(* CODESYS project Rezka.project
   Company: Plinfa
   Title: Rezka
   Author: Surmylo Serhii
   Version: 0.0.0.0

Project tree, tasks and I/O mapping:
  MyController : TM241CEC24T/U, Schneider Electric, order no. TM241CEC24T/U, version 4.0.2.20
    application Application
      task MAST (cyclic, interval 20 ms, priority 15, watchdog 100 ms x 1) calls POU_outputs_11_20, POU_outputs_21_30, POU_outputs_31_40, POU_outputs_41_50, POU_outputs_51_64, POU_outputs_drivers, POU_10_outputs_oilstation, POU_1_Utils, POU_2_TrosTolkateli, POU_3_PodvodTelezhki, POU_4_Zahvat, POU_6_HorizontalCutting, POU_7_VerticalCutting, POU_9_altivars, POU_5_Oprokidyvanie
      function HiddenPOU [ST]
      global variables GVL
      trace Trace (task MAST): POU.M_K1
      Symbols
      program POU_10_outputs_oilstation [LD]
      program POU_4_Zahvat [LD]
      program POU_1_Utils [LD]
      program POU_outputs_11_20 [LD]
      program POU_outputs_31_40 [LD]
      program POU_outputs_21_30 [LD]
      program POU_outputs_41_50 [LD]
      program POU_outputs_51_64 [LD]
      program POU_3_PodvodTelezhki [LD]
      program POU_2_TrosTolkateli [LD]
      program POU_outputs_drivers [LD]
      program POU_9_altivars [LD]
      program POU_7_VerticalCutting [LD]
      program POU_6_HorizontalCutting [LD]
      program POU_5_Oprokidyvanie [LD]
      program POU_interlock [LD]
      program POU_interlock_double [LD]
      module_unites/
        program PressTable_in [LD]
        program GrabTroll_out [LD]
        program GrabTroll_in [LD]
        program CentrTroll_in [LD]
        program TurnTroll_in [LD]
        program CentrTroll_out [LD]
        program TurnTroll_out [LD]
        program TakeTable_in [LD]
        program TakeTable_out [LD]
        program MoveTipper_in [LD]
        program MoveTipper_out [LD]
        program FixingFrame_in [LD]
        program FixingFrame_out [LD]
        program PressTable_out [LD]
        program CuttingFrame_dn [LD]
        program CuttingFrame_up [LD]
        program MovingFrame_fwd [LD]
        program MovingFrame_rev [LD]
    DI : Digital Inputs, Schneider Electric, version 4.0.2.20
        unmapped channels: IW0, IB1
    DQ : Digital Outputs, Schneider Electric, version 4.0.2.20
        unmapped channels: QW0, QB1
    Counters : Counters, Schneider Electric, version 4.0.2.20
    Pulse_Generators : Pulse Generators, Schneider Electric, version 4.0.2.20
    Cartridge_1 : Cartridge, Schneider Electric, version 4.0.2.20
    IO_Bus : IO bus - TM3, Schneider Electric, version 4.0.2.20
      Module_1 : TM3DI32K, Schneider Electric, order no. TM3DI32K, version 1.0.1.1
          input  idwModule_1_ID0 : DWORD  // ID0
          input  KM2 : BOOL  // ID0.I0
          input  KM3 : BOOL  // ID0.I1
          input  KM4 : BOOL  // ID0.I2
          input  KM7 : BOOL  // ID0.I3
          input  KM8 : BOOL  // ID0.I4
          input  KM9 : BOOL  // ID0.I5
          input  KM10 : BOOL  // ID0.I6
          input  KM11 : BOOL  // ID0.I7
          input  KM12 : BOOL  // ID0.I8
          input  KM13 : BOOL  // ID0.I9
          input  KM14 : BOOL  // ID0.I10
          input  PuskAvt : BOOL  // ID0.I11
          input  Stop : BOOL  // ID0.I12
          input  SQ1_s : BOOL  // ID0.I16
          input  SQ2_s : BOOL  // ID0.I17
          input  Kluch1_s : BOOL  // ID0.I18
          input  Vper1_s : BOOL  // ID0.I19
          input  Naz1_s : BOOL  // ID0.I20
          input  SQ3_s : BOOL  // ID0.I21
          input  SQ4_s : BOOL  // ID0.I22
          input  SQ5_s : BOOL  // ID0.I23
          input  SQ6_s : BOOL  // ID0.I24
          input  HED2_1_s : BOOL  // ID0.I25
          input  HED2_2_s : BOOL  // ID0.I26
          input  HED2_5_s : BOOL  // ID0.I29
      Module_2 : TM3DI32K, Schneider Electric, order no. TM3DI32K, version 1.0.1.1
          input  idwModule_2_ID0 : DWORD  // ID0
          input  C3B_s : BOOL  // ID0.I1
          input  C4B_s : BOOL  // ID0.I2
          input  C5B_s : BOOL  // ID0.I3
          input  C6B_s : BOOL  // ID0.I4
          input  C5C_s : BOOL  // ID0.I5
          input  C6C_s : BOOL  // ID0.I6
          input  C13B_s : BOOL  // ID0.I7
          input  C14B_s : BOOL  // ID0.I8
          input  C13C_s : BOOL  // ID0.I9
          input  C14C_s : BOOL  // ID0.I10
          input  C11B_s : BOOL  // ID0.I11
          input  C12B_s : BOOL  // ID0.I12
          input  C34_s : BOOL  // ID0.I13
          input  C3A_s : BOOL  // ID0.I14
          input  C4A_s : BOOL  // ID0.I15
          input  C5A_s : BOOL  // ID0.I16
          input  C6A_s : BOOL  // ID0.I17
          input  C5D_s : BOOL  // ID0.I18
          input  C6D_s : BOOL  // ID0.I19
          input  C13A_s : BOOL  // ID0.I20
          input  C14A_s : BOOL  // ID0.I21
          input  C13D_s : BOOL  // ID0.I22
          input  C14D_s : BOOL  // ID0.I23
          input  C11A_s : BOOL  // ID0.I24
          input  C12A_s : BOOL  // ID0.I25
          input  C17_s : BOOL  // ID0.I26
          input  C17A_s : BOOL  // ID0.I27
          input  C17B_s : BOOL  // ID0.I28
          input  C18A_s : BOOL  // ID0.I29
          input  C18B_s : BOOL  // ID0.I30
          input  C17C_s : BOOL  // ID0.I31
      Module_3 : TM3DI32K, Schneider Electric, order no. TM3DI32K, version 1.0.1.1
          input  idwModule_3_ID0 : DWORD  // ID0
          input  C17D_s : BOOL  // ID0.I0
          input  C18C_s : BOOL  // ID0.I1
          input  C18D_s : BOOL  // ID0.I2
          input  C16_s : BOOL  // ID0.I3
          input  C21_s : BOOL  // ID0.I4
          input  C22_s : BOOL  // ID0.I5
          input  C28_s : BOOL  // ID0.I6
          input  C29_s : BOOL  // ID0.I7
          input  C30_s : BOOL  // ID0.I8
          input  C31_s : BOOL  // ID0.I9
          input  C32_s : BOOL  // ID0.I10
          input  C2_s : BOOL  // ID0.I11
          input  C2A_s : BOOL  // ID0.I12
          input  C23B_s : BOOL  // ID0.I13
          input  C23C_s : BOOL  // ID0.I14
          input  C7_s : BOOL  // ID0.I15
          input  C8_s : BOOL  // ID0.I16
          input  C9_s : BOOL  // ID0.I17
          input  C15_s : BOOL  // ID0.I18
          input  C19_s : BOOL  // ID0.I19
          input  C20_s : BOOL  // ID0.I20
          input  C27_s : BOOL  // ID0.I21
          input  C33_s : BOOL  // ID0.I22
          input  C35_s : BOOL  // ID0.I23
          input  C1_s : BOOL  // ID0.I24
          input  C1A_s : BOOL  // ID0.I25
          input  C23A_s : BOOL  // ID0.I26
          input  C23D_s : BOOL  // ID0.I27
          input  C25_s : BOOL  // ID0.I28
          input  C26_s : BOOL  // ID0.I29
          input  C10_s : BOOL  // ID0.I31
      Module_4 : TM3DI32K, Schneider Electric, order no. TM3DI32K, version 1.0.1.1
          input  idwModule_4_ID0 : DWORD  // ID0
          input  SQ10_s : BOOL  // ID0.I0
          input  SQ11_s : BOOL  // ID0.I1
          input  Kluch2_s : BOOL  // ID0.I2
          input  Vper2_s : BOOL  // ID0.I3
          input  Naz2_s : BOOL  // ID0.I4
          input  SQ12_s : BOOL  // ID0.I5
          input  SQ13_s : BOOL  // ID0.I6
          input  SQ14_s : BOOL  // ID0.I7
          input  Kluch3_s : BOOL  // ID0.I8
          input  Vper3_s : BOOL  // ID0.I9
          input  Naz3_s : BOOL  // ID0.I10
          input  SQ15_s : BOOL  // ID0.I11
          input  SQ16_s : BOOL  // ID0.I12
          input  SQ17_s : BOOL  // ID0.I13
          input  SQ18_s : BOOL  // ID0.I14
          input  SQ19_s : BOOL  // ID0.I15
          input  C21shtrih_s : BOOL  // ID0.I20
          input  C22shtrih_s : BOOL  // ID0.I21
      Module_5 : TM3DQ32TK, Schneider Electric, order no. TM3DQ32TK, version 1.0.1.1
          output KL1 : BOOL  // QD0.Q0
          output KL2 : BOOL  // QD0.Q1
          output KL3 : BOOL  // QD0.Q2
          output KL4 : BOOL  // QD0.Q3
          output KL5 : BOOL  // QD0.Q4
          output KL6 : BOOL  // QD0.Q5
          output KL7 : BOOL  // QD0.Q6
          output KL8 : BOOL  // QD0.Q7
          output KL9 : BOOL  // QD0.Q8
          output KL10 : BOOL  // QD0.Q9
          output KL11 : BOOL  // QD0.Q10
          output KL12 : BOOL  // QD0.Q11
          output KL13 : BOOL  // QD0.Q12
          output KL14 : BOOL  // QD0.Q13
          output KL15 : BOOL  // QD0.Q14
          output KL16 : BOOL  // QD0.Q15
          output KL17 : BOOL  // QD0.Q16
          output KL18 : BOOL  // QD0.Q17
          output KL19 : BOOL  // QD0.Q18
          output KL20 : BOOL  // QD0.Q19
          output KL21 : BOOL  // QD0.Q20
          output KL22 : BOOL  // QD0.Q21
          output KL23 : BOOL  // QD0.Q22
          output KL24 : BOOL  // QD0.Q23
          output KL25 : BOOL  // QD0.Q24
          output KL26 : BOOL  // QD0.Q25
          output KL27 : BOOL  // QD0.Q26
          output KL28 : BOOL  // QD0.Q27
          output KL29 : BOOL  // QD0.Q28
          output KL30 : BOOL  // QD0.Q29
          output KL31 : BOOL  // QD0.Q30
          output KL32 : BOOL  // QD0.Q31
          unmapped channels: QD0
      Module_6 : TM3DQ32TK, Schneider Electric, order no. TM3DQ32TK, version 1.0.1.1
          output KL33 : BOOL  // QD0.Q0
          output KL34 : BOOL  // QD0.Q1
          output KL35 : BOOL  // QD0.Q2
          output KL36 : BOOL  // QD0.Q3
          output KL37 : BOOL  // QD0.Q4
          output KL38 : BOOL  // QD0.Q5
          output KL39 : BOOL  // QD0.Q6
          output KL40 : BOOL  // QD0.Q7
          output KL41 : BOOL  // QD0.Q8
          output KL42 : BOOL  // QD0.Q9
          output KL43 : BOOL  // QD0.Q10
          output KL44 : BOOL  // QD0.Q11
          output KL45 : BOOL  // QD0.Q12
          output KL46 : BOOL  // QD0.Q13
          output KL47 : BOOL  // QD0.Q14
          output KL48 : BOOL  // QD0.Q15
          output KL49 : BOOL  // QD0.Q16
          output KL50 : BOOL  // QD0.Q17
          output KL51 : BOOL  // QD0.Q18
          output KL52 : BOOL  // QD0.Q19
          output KL53 : BOOL  // QD0.Q20
          output KL54 : BOOL  // QD0.Q21
          output KL55 : BOOL  // QD0.Q22
          output KL56 : BOOL  // QD0.Q23
          output KL57 : BOOL  // QD0.Q24
          output KL58 : BOOL  // QD0.Q25
          output KL59 : BOOL  // QD0.Q26
          output KL60 : BOOL  // QD0.Q27
          output KL61 : BOOL  // QD0.Q28
          output KL62 : BOOL  // QD0.Q29
          output KL63 : BOOL  // QD0.Q30
          output KL64 : BOOL  // QD0.Q31
          unmapped channels: QD0
    COM_Bus : COM bus, Schneider Electric, version 4.0.2.20
    Ethernet_1 : Ethernet Network, Schneider Electric, version 4.0.2.20
        settings: IPAddress = [192, 168, 49, 90]; SubnetMask = [255, 255, 255, 0]; GatewayAddress = [192, 168, 49, 1]; DeviceName = 'sch_cutter'; WebServer = TRUE; FTP Server = FALSE; SoMachine Protocol = TRUE; Modbus Server = TRUE; NetManage Protocol = TRUE; SNMP protocol = TRUE; Enable Routing = FALSE; WebVisu protocol = FALSE
      ModbusTCP_Slave_Device : ModbusTCP Slave Device, Schneider Electric, version 3.5.2.3
          settings: IPMasterAddress = [192, 168, 0, 90]
          unmapped channels: Inputs, Outputs
    Serial_Line_1 : Serial line, Schneider Electric, version 4.0.2.20
      SoMachine_Network_Manager : SoMachine-Network Manager, Schneider Electric, version 4.0.0.2
    Serial_Line_2 : Serial line, Schneider Electric, version 4.0.2.20
      Modbus_Manager : Modbus Manager, Schneider Electric, version 4.0.0.2
    CAN_1 : CANopen bus, Schneider Electric, version 4.0.2.20
      CANopen_Performance : CANopen Performance, Schneider Electric, order no. 1806, version 3.0.1.22
          settings: ConfigVersion = 50659584
        Altivar_71_0 : Altivar 71, Schneider Electric, order no. 71, version 4.4.5.0
            settings: General Options.Optional Device = TRUE; General Options.Reset Node = TRUE; NODEIDSAVED = 1; SDO Timeout = 1000000; Explicit Deactivate PDOs = TRUE; EXPERTSETTINGS = True; Heartbeat-Producer Time = 300; PDO 16#1400.COBID = 16#0201; Settings.COBID = 16#0181; Settings.Transmission Type = 16#FF; Settings.available PDO-Parameter.Inhibit Time available = TRUE; Settings.available PDO-Parameter.Event Timer available = TRUE; Settings.Inhibit Time = 30; Settings.Event Timer = 1000; Generic COBID = '$NODEID+16#0180'; Heartbeat-Consuming1.Heartbeat-Time = 300 ms; Controlword.Subindex = 16#00; Frequency ref..Index = 16#2002; Frequency ref..Subindex = 16#04; Frequency ref..ObjectLength = 16; Motor current.Index = 16#2002; Motor current.Subindex = 16#05; Motor current.ObjectLength = 16; Output frequency.Index = 16#2002; Output frequency.Subindex = 16#03; Output frequency.ObjectLength = 16; Error Code.Index = 16#603F; Error Code.Subindex = 16#00; Error Code.ObjectLength = 16; Statusword.Index = 16#6041; Statusword.Subindex = 16#00; Statusword.ObjectLength = 16; SDO List.Set Guardtime.Index = 16#100C; SDO List.Set Guardtime.Subindex = 16#00; SDO List.Set Guardtime.Value = 16#00000000; SDO List.Set Guardtime.Size = 16; SDO List.Set Guardtime.AbortIfError = FALSE; SDO List.Set Guardtime.JumpToLine = FALSE; SDO List.Set Guardtime.Line = 0; SDO List.Set Lifetime.Index = 16#100D;
              SDO List.Set Lifetime.Subindex = 16#00; SDO List.Set Lifetime.Value = 16#00000000; SDO List.Set Lifetime.Size = 8; SDO List.Set Lifetime.AbortIfError = FALSE; SDO List.Set Lifetime.JumpToLine = FALSE; SDO List.Set Lifetime.Line = 0; SDO List.Set Heartbeat Consumer.Index = 16#1016; SDO List.Set Heartbeat Consumer.Subindex = 16#01; SDO List.Set Heartbeat Consumer.Value = 16#007F012C; SDO List.Set Heartbeat Consumer.Size = 32; SDO List.Set Heartbeat Consumer.AbortIfError = FALSE; SDO List.Set Heartbeat Consumer.JumpToLine = FALSE; SDO List.Set Heartbeat Consumer.Line = 0; SDO List.Set Heartbeat Producer.Index = 16#1017; SDO List.Set Heartbeat Producer.Subindex = 16#00; SDO List.Set Heartbeat Producer.Value = 16#0000012C; SDO List.Set Heartbeat Producer.Size = 16; SDO List.Set Heartbeat Producer.AbortIfError = FALSE; SDO List.Set Heartbeat Producer.JumpToLine = FALSE; SDO List.Set Heartbeat Producer.Line = 0; SDO List.Disable PDO.Index = 16#1400; SDO List.Disable PDO.Subindex = 16#01; SDO List.Disable PDO.Value = 16#80000201; SDO List.Disable PDO.Size = 32; SDO List.Disable PDO.AbortIfError = FALSE; SDO List.Disable PDO.JumpToLine = FALSE; SDO List.Disable PDO.Line = 0; SDO List.Set transmission type.Index = 16#1400; SDO List.Set transmission type.Subindex = 16#02; SDO List.Set transmission type.Value = 16#FF; SDO List.Set transmission type.Size = 8; SDO List.Set transmission type.AbortIfError = FALSE; SDO List.Set transmission type.JumpToLine = FALSE; SDO List.Set transmission type.Line = 0; SDO List.Clear pdo mapping.Index = 16#1600; SDO List.Clear pdo mapping.Subindex = 16#00; SDO List.Clear pdo mapping.Value = 16#0; SDO List.Clear pdo mapping.Size = 8; SDO List.Clear pdo mapping.AbortIfError = FALSE; SDO List.Clear pdo mapping.JumpToLine = FALSE;
              SDO List.Clear pdo mapping.Line = 0; SDO List.Set Mapping.Index = 16#1600; SDO List.Set Mapping.Subindex = 16#01; SDO List.Set Mapping.Value = 16#60400010; SDO List.Set Mapping.Size = 32; SDO List.Set Mapping.AbortIfError = FALSE; SDO List.Set Mapping.JumpToLine = FALSE; SDO List.Set Mapping.Line = 0; SDO List.Set Mapping.Index = 16#1600; SDO List.Set Mapping.Subindex = 16#02; SDO List.Set Mapping.Value = 16#20020410; SDO List.Set Mapping.Size = 32; SDO List.Set Mapping.AbortIfError = FALSE; SDO List.Set Mapping.JumpToLine = FALSE; SDO List.Set Mapping.Line = 0; SDO List.Set Mapping.Index = 16#1600; SDO List.Set Mapping.Subindex = 16#03; SDO List.Set Mapping.Value = 16#20020510; SDO List.Set Mapping.Size = 32; SDO List.Set Mapping.AbortIfError = FALSE; SDO List.Set Mapping.JumpToLine = FALSE; SDO List.Set Mapping.Line = 0; SDO List.Set Mapping.Index = 16#1600; SDO List.Set Mapping.Subindex = 16#04; SDO List.Set Mapping.Value = 16#20020310; SDO List.Set Mapping.Size = 32; SDO List.Set Mapping.AbortIfError = FALSE; SDO List.Set Mapping.JumpToLine = FALSE; SDO List.Set Mapping.Line = 0; SDO List.Set number of pdos.Index = 16#1600; SDO List.Set number of pdos.Subindex = 16#00; SDO List.Set number of pdos.Value = 16#04; SDO List.Set number of pdos.Size = 8; SDO List.Set number of pdos.AbortIfError = FALSE; SDO List.Set number of pdos.JumpToLine = FALSE; SDO List.Set number of pdos.Line = 0; SDO List.Set and enable COB-ID.Index = 16#1400; SDO List.Set and enable COB-ID.Subindex = 16#01; SDO List.Set and enable COB-ID.Value = 16#00000201; SDO List.Set and enable COB-ID.Size = 32;
              SDO List.Set and enable COB-ID.AbortIfError = FALSE; SDO List.Set and enable COB-ID.JumpToLine = FALSE; SDO List.Set and enable COB-ID.Line = 0; SDO List.Disable PDO.Index = 16#1800; SDO List.Disable PDO.Subindex = 16#01; SDO List.Disable PDO.Value = 16#80000181; SDO List.Disable PDO.Size = 32; SDO List.Disable PDO.AbortIfError = FALSE; SDO List.Disable PDO.JumpToLine = FALSE; SDO List.Disable PDO.Line = 0; SDO List.Set transmission type.Index = 16#1800; SDO List.Set transmission type.Subindex = 16#02; SDO List.Set transmission type.Value = 16#FF; SDO List.Set transmission type.Size = 8; SDO List.Set transmission type.AbortIfError = FALSE; SDO List.Set transmission type.JumpToLine = FALSE; SDO List.Set transmission type.Line = 0; SDO List.Set inhibit time.Index = 16#1800; SDO List.Set inhibit time.Subindex = 16#03; SDO List.Set inhibit time.Value = 16#001E; SDO List.Set inhibit time.Size = 16; SDO List.Set inhibit time.AbortIfError = FALSE; SDO List.Set inhibit time.JumpToLine = FALSE; SDO List.Set inhibit time.Line = 0; SDO List.Set event time.Index = 16#1800; SDO List.Set event time.Subindex = 16#05; SDO List.Set event time.Value = 16#03E8; SDO List.Set event time.Size = 16; SDO List.Set event time.AbortIfError = FALSE; SDO List.Set event time.JumpToLine = FALSE; SDO List.Set event time.Line = 0; SDO List.Clear pdo mapping.Index = 16#1A00; SDO List.Clear pdo mapping.Subindex = 16#00; SDO List.Clear pdo mapping.Value = 16#0; SDO List.Clear pdo mapping.Size = 8; SDO List.Clear pdo mapping.AbortIfError = FALSE; SDO List.Clear pdo mapping.JumpToLine = FALSE; SDO List.Clear pdo mapping.Line = 0; SDO List.Set Mapping.Index = 16#1A00; SDO List.Set Mapping.Subindex = 16#01;
              SDO List.Set Mapping.Value = 16#603F0010; SDO List.Set Mapping.Size = 32; SDO List.Set Mapping.AbortIfError = FALSE; SDO List.Set Mapping.JumpToLine = FALSE; SDO List.Set Mapping.Line = 0; SDO List.Set Mapping.Index = 16#1A00; SDO List.Set Mapping.Subindex = 16#02; SDO List.Set Mapping.Value = 16#60410010; SDO List.Set Mapping.Size = 32; SDO List.Set Mapping.AbortIfError = FALSE; SDO List.Set Mapping.JumpToLine = FALSE; SDO List.Set Mapping.Line = 0; SDO List.Set number of pdos.Index = 16#1A00; SDO List.Set number of pdos.Subindex = 16#00; SDO List.Set number of pdos.Value = 16#02; SDO List.Set number of pdos.Size = 8; SDO List.Set number of pdos.AbortIfError = FALSE; SDO List.Set number of pdos.JumpToLine = FALSE; SDO List.Set number of pdos.Line = 0; SDO List.Set and enable COB-ID.Index = 16#1800; SDO List.Set and enable COB-ID.Subindex = 16#01; SDO List.Set and enable COB-ID.Value = 16#00000181; SDO List.Set and enable COB-ID.Size = 32; SDO List.Set and enable COB-ID.AbortIfError = FALSE; SDO List.Set and enable COB-ID.JumpToLine = FALSE; SDO List.Set and enable COB-ID.Line = 0; ConfigVersion = 50659584
            output altivar_0_Controlword : UINT  // Controlword
            input  altivar_0_Statusword : UINT  // Statusword
            unmapped channels: Frequency ref., Motor current, Output frequency, Error Code
        Altivar_71_1 : Altivar 71, Schneider Electric, order no. 71, version 4.4.5.0
            settings: General Options.Optional Device = TRUE; General Options.Reset Node = TRUE; NODEIDSAVED = 2; SDO Timeout = 1000000; Explicit Deactivate PDOs = FALSE; EXPERTSETTINGS = FALSE; Emergency-General Parameters.Emergency COBID = 16#82; Heartbeat-Producer Time = 200; PDO 16#1400.COBID = 16#80000202; PDO 16#1401.COBID = 16#0302; PDO 16#1402.COBID = 16#80000402; PDO 16#1800.COBID = 16#0182; PDO 16#1801.COBID = 16#0282; PDO 16#1802.COBID = 16#80000382; Heartbeat-Consuming1.Heartbeat-Time = 300 ms; Controlword.Subindex = 16#00; Target Velocity.Subindex = 16#00; Controlword.Subindex = 16#00; HMI Frequency ref..Subindex = 16#03; Received PD03-1.Subindex = 16#02; Received PD03-2.Subindex = 16#03; Received PD03-3.Subindex = 16#04; Received PD03-4.Subindex = 16#05; OL1R.Subindex = 16#0D; Statusword.Subindex = 16#00; ETI state word.Subindex = 16#07; Control Effort.Subindex = 16#00; IL1R.Subindex = 16#03; Transmit PDO3-1.Subindex = 16#0C; Transmit PDO3-2.Subindex = 16#0D; Transmit PDO3-3.Subindex = 16#0E; Transmit PDO3-4.Subindex = 16#0F; SDO List.Set Guardtime.Index = 16#100C; SDO List.Set Guardtime.Subindex = 16#00; SDO List.Set Guardtime.Value = 16#00000000; SDO List.Set Guardtime.Size = 16; SDO List.Set Guardtime.AbortIfError = FALSE; SDO List.Set Guardtime.JumpToLine = FALSE; SDO List.Set Guardtime.Line = 0; SDO List.Set Lifetime.Index = 16#100D;
              SDO List.Set Lifetime.Subindex = 16#00; SDO List.Set Lifetime.Value = 16#00000000; SDO List.Set Lifetime.Size = 8; SDO List.Set Lifetime.AbortIfError = FALSE; SDO List.Set Lifetime.JumpToLine = FALSE; SDO List.Set Lifetime.Line = 0; SDO List.Set Heartbeat Consumer.Index = 16#1016; SDO List.Set Heartbeat Consumer.Subindex = 16#01; SDO List.Set Heartbeat Consumer.Value = 16#007F012C; SDO List.Set Heartbeat Consumer.Size = 32; SDO List.Set Heartbeat Consumer.AbortIfError = FALSE; SDO List.Set Heartbeat Consumer.JumpToLine = FALSE; SDO List.Set Heartbeat Consumer.Line = 0; SDO List.Set Heartbeat Producer.Index = 16#1017; SDO List.Set Heartbeat Producer.Subindex = 16#00; SDO List.Set Heartbeat Producer.Value = 16#000000C8; SDO List.Set Heartbeat Producer.Size = 16; SDO List.Set Heartbeat Producer.AbortIfError = FALSE; SDO List.Set Heartbeat Producer.JumpToLine = FALSE; SDO List.Set Heartbeat Producer.Line = 0; SDO List.Disable PDO.Index = 16#1401; SDO List.Disable PDO.Subindex = 16#01; SDO List.Disable PDO.Value = 16#80000302; SDO List.Disable PDO.Size = 32; SDO List.Disable PDO.AbortIfError = FALSE; SDO List.Disable PDO.JumpToLine = FALSE; SDO List.Disable PDO.Line = 0; SDO List.Set transmission type.Index = 16#1401; SDO List.Set transmission type.Subindex = 16#02; SDO List.Set transmission type.Value = 16#FF; SDO List.Set transmission type.Size = 8; SDO List.Set transmission type.AbortIfError = FALSE; SDO List.Set transmission type.JumpToLine = FALSE; SDO List.Set transmission type.Line = 0; SDO List.Clear pdo mapping.Index = 16#1601; SDO List.Clear pdo mapping.Subindex = 16#00; SDO List.Clear pdo mapping.Value = 16#0; SDO List.Clear pdo mapping.Size = 8; SDO List.Clear pdo mapping.AbortIfError = FALSE; SDO List.Clear pdo mapping.JumpToLine = FALSE;
              SDO List.Clear pdo mapping.Line = 0; SDO List.Set Mapping.Index = 16#1601; SDO List.Set Mapping.Subindex = 16#01; SDO List.Set Mapping.Value = 16#60400010; SDO List.Set Mapping.Size = 32; SDO List.Set Mapping.AbortIfError = FALSE; SDO List.Set Mapping.JumpToLine = FALSE; SDO List.Set Mapping.Line = 0; SDO List.Set Mapping.Index = 16#1601; SDO List.Set Mapping.Subindex = 16#02; SDO List.Set Mapping.Value = 16#20370310; SDO List.Set Mapping.Size = 32; SDO List.Set Mapping.AbortIfError = FALSE; SDO List.Set Mapping.JumpToLine = FALSE; SDO List.Set Mapping.Line = 0; SDO List.Set number of pdos.Index = 16#1601; SDO List.Set number of pdos.Subindex = 16#00; SDO List.Set number of pdos.Value = 16#02; SDO List.Set number of pdos.Size = 8; SDO List.Set number of pdos.AbortIfError = FALSE; SDO List.Set number of pdos.JumpToLine = FALSE; SDO List.Set number of pdos.Line = 0; SDO List.Set and enable COB-ID.Index = 16#1401; SDO List.Set and enable COB-ID.Subindex = 16#01; SDO List.Set and enable COB-ID.Value = 16#00000302; SDO List.Set and enable COB-ID.Size = 32; SDO List.Set and enable COB-ID.AbortIfError = FALSE; SDO List.Set and enable COB-ID.JumpToLine = FALSE; SDO List.Set and enable COB-ID.Line = 0; SDO List.Disable PDO.Index = 16#1800; SDO List.Disable PDO.Subindex = 16#01; SDO List.Disable PDO.Value = 16#80000182; SDO List.Disable PDO.Size = 32; SDO List.Disable PDO.AbortIfError = FALSE; SDO List.Disable PDO.JumpToLine = FALSE; SDO List.Disable PDO.Line = 0; SDO List.Set transmission type.Index = 16#1800; SDO List.Set transmission type.Subindex = 16#02; SDO List.Set transmission type.Value = 16#FF; SDO List.Set transmission type.Size = 8;
              SDO List.Set transmission type.AbortIfError = FALSE; SDO List.Set transmission type.JumpToLine = FALSE; SDO List.Set transmission type.Line = 0; SDO List.Set inhibit time.Index = 16#1800; SDO List.Set inhibit time.Subindex = 16#03; SDO List.Set inhibit time.Value = 16#001E; SDO List.Set inhibit time.Size = 16; SDO List.Set inhibit time.AbortIfError = FALSE; SDO List.Set inhibit time.JumpToLine = FALSE; SDO List.Set inhibit time.Line = 0; SDO List.Set event time.Index = 16#1800; SDO List.Set event time.Subindex = 16#05; SDO List.Set event time.Value = 16#03E8; SDO List.Set event time.Size = 16; SDO List.Set event time.AbortIfError = FALSE; SDO List.Set event time.JumpToLine = FALSE; SDO List.Set event time.Line = 0; SDO List.Clear pdo mapping.Index = 16#1A00; SDO List.Clear pdo mapping.Subindex = 16#00; SDO List.Clear pdo mapping.Value = 16#0; SDO List.Clear pdo mapping.Size = 8; SDO List.Clear pdo mapping.AbortIfError = FALSE; SDO List.Clear pdo mapping.JumpToLine = FALSE; SDO List.Clear pdo mapping.Line = 0; SDO List.Set Mapping.Index = 16#1A00; SDO List.Set Mapping.Subindex = 16#01; SDO List.Set Mapping.Value = 16#20160D10; SDO List.Set Mapping.Size = 32; SDO List.Set Mapping.AbortIfError = FALSE; SDO List.Set Mapping.JumpToLine = FALSE; SDO List.Set Mapping.Line = 0; SDO List.Set number of pdos.Index = 16#1A00; SDO List.Set number of pdos.Subindex = 16#00; SDO List.Set number of pdos.Value = 16#01; SDO List.Set number of pdos.Size = 8; SDO List.Set number of pdos.AbortIfError = FALSE; SDO List.Set number of pdos.JumpToLine = FALSE; SDO List.Set number of pdos.Line = 0; SDO List.Set and enable COB-ID.Index = 16#1800; SDO List.Set and enable COB-ID.Subindex = 16#01;
              SDO List.Set and enable COB-ID.Value = 16#00000182; SDO List.Set and enable COB-ID.Size = 32; SDO List.Set and enable COB-ID.AbortIfError = FALSE; SDO List.Set and enable COB-ID.JumpToLine = FALSE; SDO List.Set and enable COB-ID.Line = 0; SDO List.Disable PDO.Index = 16#1801; SDO List.Disable PDO.Subindex = 16#01; SDO List.Disable PDO.Value = 16#80000282; SDO List.Disable PDO.Size = 32; SDO List.Disable PDO.AbortIfError = FALSE; SDO List.Disable PDO.JumpToLine = FALSE; SDO List.Disable PDO.Line = 0; SDO List.Set transmission type.Index = 16#1801; SDO List.Set transmission type.Subindex = 16#02; SDO List.Set transmission type.Value = 16#FF; SDO List.Set transmission type.Size = 8; SDO List.Set transmission type.AbortIfError = FALSE; SDO List.Set transmission type.JumpToLine = FALSE; SDO List.Set transmission type.Line = 0; SDO List.Set inhibit time.Index = 16#1801; SDO List.Set inhibit time.Subindex = 16#03; SDO List.Set inhibit time.Value = 16#001E; SDO List.Set inhibit time.Size = 16; SDO List.Set inhibit time.AbortIfError = FALSE; SDO List.Set inhibit time.JumpToLine = FALSE; SDO List.Set inhibit time.Line = 0; SDO List.Set event time.Index = 16#1801; SDO List.Set event time.Subindex = 16#05; SDO List.Set event time.Value = 16#03E8; SDO List.Set event time.Size = 16; SDO List.Set event time.AbortIfError = FALSE; SDO List.Set event time.JumpToLine = FALSE; SDO List.Set event time.Line = 0; SDO List.Clear pdo mapping.Index = 16#1A01; SDO List.Clear pdo mapping.Subindex = 16#00; SDO List.Clear pdo mapping.Value = 16#0; SDO List.Clear pdo mapping.Size = 8; SDO List.Clear pdo mapping.AbortIfError = FALSE; SDO List.Clear pdo mapping.JumpToLine = FALSE; SDO List.Clear pdo mapping.Line = 0;
              SDO List.Set Mapping.Index = 16#1A01; SDO List.Set Mapping.Subindex = 16#01; SDO List.Set Mapping.Value = 16#60410010; SDO List.Set Mapping.Size = 32; SDO List.Set Mapping.AbortIfError = FALSE; SDO List.Set Mapping.JumpToLine = FALSE; SDO List.Set Mapping.Line = 0; SDO List.Set Mapping.Index = 16#1A01; SDO List.Set Mapping.Subindex = 16#02; SDO List.Set Mapping.Value = 16#20020710; SDO List.Set Mapping.Size = 32; SDO List.Set Mapping.AbortIfError = FALSE; SDO List.Set Mapping.JumpToLine = FALSE; SDO List.Set Mapping.Line = 0; SDO List.Set Mapping.Index = 16#1A01; SDO List.Set Mapping.Subindex = 16#03; SDO List.Set Mapping.Value = 16#60440010; SDO List.Set Mapping.Size = 32; SDO List.Set Mapping.AbortIfError = FALSE; SDO List.Set Mapping.JumpToLine = FALSE; SDO List.Set Mapping.Line = 0; SDO List.Set Mapping.Index = 16#1A01; SDO List.Set Mapping.Subindex = 16#04; SDO List.Set Mapping.Value = 16#20160310; SDO List.Set Mapping.Size = 32; SDO List.Set Mapping.AbortIfError = FALSE; SDO List.Set Mapping.JumpToLine = FALSE; SDO List.Set Mapping.Line = 0; SDO List.Set number of pdos.Index = 16#1A01; SDO List.Set number of pdos.Subindex = 16#00; SDO List.Set number of pdos.Value = 16#04; SDO List.Set number of pdos.Size = 8; SDO List.Set number of pdos.AbortIfError = FALSE; SDO List.Set number of pdos.JumpToLine = FALSE; SDO List.Set number of pdos.Line = 0; SDO List.Set and enable COB-ID.Index = 16#1801; SDO List.Set and enable COB-ID.Subindex = 16#01; SDO List.Set and enable COB-ID.Value = 16#00000282; SDO List.Set and enable COB-ID.Size = 32; SDO List.Set and enable COB-ID.AbortIfError = FALSE;
              SDO List.Set and enable COB-ID.JumpToLine = FALSE; SDO List.Set and enable COB-ID.Line = 0; ConfigVersion = 50659584
            output altivar_1_Controlword : UINT  // Controlword
            output altivar_1_HMI_Frequency_ref : INT  // HMI Frequency ref.
            input  altivar_1_OL1R : UINT  // OL1R
            input  altivar_1_Statusword : UINT  // Statusword
            input  altivar_1_ETI_state_word : UINT  // ETI state word
            input  altivar_1_Control_Effort : INT  // Control Effort
            input  altivar_1_IL1R : UINT  // IL1R
        Altivar_71_2 : Altivar 71, Schneider Electric, order no. 71, version 4.4.5.0
            settings: General Options.Optional Device = TRUE; General Options.Reset Node = TRUE; NODEIDSAVED = 3; SDO Timeout = 1000000; Explicit Deactivate PDOs = FALSE; EXPERTSETTINGS = FALSE; Emergency-General Parameters.Emergency COBID = 16#83; Heartbeat-Producer Time = 200; PDO 16#1400.COBID = 16#80000203; PDO 16#1401.COBID = 16#0303; PDO 16#1402.COBID = 16#80000403; PDO 16#1800.COBID = 16#0183; PDO 16#1801.COBID = 16#0283; PDO 16#1802.COBID = 16#80000383; Heartbeat-Consuming1.Heartbeat-Time = 300 ms; Controlword.Subindex = 16#00; Target Velocity.Subindex = 16#00; Controlword.Subindex = 16#00; HMI Frequency ref..Subindex = 16#03; Received PD03-1.Subindex = 16#02; Received PD03-2.Subindex = 16#03; Received PD03-3.Subindex = 16#04; Received PD03-4.Subindex = 16#05; OL1R.Subindex = 16#0D; Statusword.Subindex = 16#00; ETI state word.Subindex = 16#07; Control Effort.Subindex = 16#00; IL1R.Subindex = 16#03; Transmit PDO3-1.Subindex = 16#0C; Transmit PDO3-2.Subindex = 16#0D; Transmit PDO3-3.Subindex = 16#0E; Transmit PDO3-4.Subindex = 16#0F; SDO List.Set Guardtime.Index = 16#100C; SDO List.Set Guardtime.Subindex = 16#00; SDO List.Set Guardtime.Value = 16#00000000; SDO List.Set Guardtime.Size = 16; SDO List.Set Guardtime.AbortIfError = FALSE; SDO List.Set Guardtime.JumpToLine = FALSE; SDO List.Set Guardtime.Line = 0; SDO List.Set Lifetime.Index = 16#100D;
              SDO List.Set Lifetime.Subindex = 16#00; SDO List.Set Lifetime.Value = 16#00000000; SDO List.Set Lifetime.Size = 8; SDO List.Set Lifetime.AbortIfError = FALSE; SDO List.Set Lifetime.JumpToLine = FALSE; SDO List.Set Lifetime.Line = 0; SDO List.Set Heartbeat Consumer.Index = 16#1016; SDO List.Set Heartbeat Consumer.Subindex = 16#01; SDO List.Set Heartbeat Consumer.Value = 16#007F012C; SDO List.Set Heartbeat Consumer.Size = 32; SDO List.Set Heartbeat Consumer.AbortIfError = FALSE; SDO List.Set Heartbeat Consumer.JumpToLine = FALSE; SDO List.Set Heartbeat Consumer.Line = 0; SDO List.Set Heartbeat Producer.Index = 16#1017; SDO List.Set Heartbeat Producer.Subindex = 16#00; SDO List.Set Heartbeat Producer.Value = 16#000000C8; SDO List.Set Heartbeat Producer.Size = 16; SDO List.Set Heartbeat Producer.AbortIfError = FALSE; SDO List.Set Heartbeat Producer.JumpToLine = FALSE; SDO List.Set Heartbeat Producer.Line = 0; SDO List.Disable PDO.Index = 16#1401; SDO List.Disable PDO.Subindex = 16#01; SDO List.Disable PDO.Value = 16#80000303; SDO List.Disable PDO.Size = 32; SDO List.Disable PDO.AbortIfError = FALSE; SDO List.Disable PDO.JumpToLine = FALSE; SDO List.Disable PDO.Line = 0; SDO List.Set transmission type.Index = 16#1401; SDO List.Set transmission type.Subindex = 16#02; SDO List.Set transmission type.Value = 16#FF; SDO List.Set transmission type.Size = 8; SDO List.Set transmission type.AbortIfError = FALSE; SDO List.Set transmission type.JumpToLine = FALSE; SDO List.Set transmission type.Line = 0; SDO List.Clear pdo mapping.Index = 16#1601; SDO List.Clear pdo mapping.Subindex = 16#00; SDO List.Clear pdo mapping.Value = 16#0; SDO List.Clear pdo mapping.Size = 8; SDO List.Clear pdo mapping.AbortIfError = FALSE; SDO List.Clear pdo mapping.JumpToLine = FALSE;
              SDO List.Clear pdo mapping.Line = 0; SDO List.Set Mapping.Index = 16#1601; SDO List.Set Mapping.Subindex = 16#01; SDO List.Set Mapping.Value = 16#60400010; SDO List.Set Mapping.Size = 32; SDO List.Set Mapping.AbortIfError = FALSE; SDO List.Set Mapping.JumpToLine = FALSE; SDO List.Set Mapping.Line = 0; SDO List.Set Mapping.Index = 16#1601; SDO List.Set Mapping.Subindex = 16#02; SDO List.Set Mapping.Value = 16#20370310; SDO List.Set Mapping.Size = 32; SDO List.Set Mapping.AbortIfError = FALSE; SDO List.Set Mapping.JumpToLine = FALSE; SDO List.Set Mapping.Line = 0; SDO List.Set number of pdos.Index = 16#1601; SDO List.Set number of pdos.Subindex = 16#00; SDO List.Set number of pdos.Value = 16#02; SDO List.Set number of pdos.Size = 8; SDO List.Set number of pdos.AbortIfError = FALSE; SDO List.Set number of pdos.JumpToLine = FALSE; SDO List.Set number of pdos.Line = 0; SDO List.Set and enable COB-ID.Index = 16#1401; SDO List.Set and enable COB-ID.Subindex = 16#01; SDO List.Set and enable COB-ID.Value = 16#00000303; SDO List.Set and enable COB-ID.Size = 32; SDO List.Set and enable COB-ID.AbortIfError = FALSE; SDO List.Set and enable COB-ID.JumpToLine = FALSE; SDO List.Set and enable COB-ID.Line = 0; SDO List.Disable PDO.Index = 16#1800; SDO List.Disable PDO.Subindex = 16#01; SDO List.Disable PDO.Value = 16#80000183; SDO List.Disable PDO.Size = 32; SDO List.Disable PDO.AbortIfError = FALSE; SDO List.Disable PDO.JumpToLine = FALSE; SDO List.Disable PDO.Line = 0; SDO List.Set transmission type.Index = 16#1800; SDO List.Set transmission type.Subindex = 16#02; SDO List.Set transmission type.Value = 16#FF; SDO List.Set transmission type.Size = 8;
              SDO List.Set transmission type.AbortIfError = FALSE; SDO List.Set transmission type.JumpToLine = FALSE; SDO List.Set transmission type.Line = 0; SDO List.Set inhibit time.Index = 16#1800; SDO List.Set inhibit time.Subindex = 16#03; SDO List.Set inhibit time.Value = 16#001E; SDO List.Set inhibit time.Size = 16; SDO List.Set inhibit time.AbortIfError = FALSE; SDO List.Set inhibit time.JumpToLine = FALSE; SDO List.Set inhibit time.Line = 0; SDO List.Set event time.Index = 16#1800; SDO List.Set event time.Subindex = 16#05; SDO List.Set event time.Value = 16#03E8; SDO List.Set event time.Size = 16; SDO List.Set event time.AbortIfError = FALSE; SDO List.Set event time.JumpToLine = FALSE; SDO List.Set event time.Line = 0; SDO List.Clear pdo mapping.Index = 16#1A00; SDO List.Clear pdo mapping.Subindex = 16#00; SDO List.Clear pdo mapping.Value = 16#0; SDO List.Clear pdo mapping.Size = 8; SDO List.Clear pdo mapping.AbortIfError = FALSE; SDO List.Clear pdo mapping.JumpToLine = FALSE; SDO List.Clear pdo mapping.Line = 0; SDO List.Set Mapping.Index = 16#1A00; SDO List.Set Mapping.Subindex = 16#01; SDO List.Set Mapping.Value = 16#20160D10; SDO List.Set Mapping.Size = 32; SDO List.Set Mapping.AbortIfError = FALSE; SDO List.Set Mapping.JumpToLine = FALSE; SDO List.Set Mapping.Line = 0; SDO List.Set number of pdos.Index = 16#1A00; SDO List.Set number of pdos.Subindex = 16#00; SDO List.Set number of pdos.Value = 16#01; SDO List.Set number of pdos.Size = 8; SDO List.Set number of pdos.AbortIfError = FALSE; SDO List.Set number of pdos.JumpToLine = FALSE; SDO List.Set number of pdos.Line = 0; SDO List.Set and enable COB-ID.Index = 16#1800; SDO List.Set and enable COB-ID.Subindex = 16#01;
              SDO List.Set and enable COB-ID.Value = 16#00000183; SDO List.Set and enable COB-ID.Size = 32; SDO List.Set and enable COB-ID.AbortIfError = FALSE; SDO List.Set and enable COB-ID.JumpToLine = FALSE; SDO List.Set and enable COB-ID.Line = 0; SDO List.Disable PDO.Index = 16#1801; SDO List.Disable PDO.Subindex = 16#01; SDO List.Disable PDO.Value = 16#80000283; SDO List.Disable PDO.Size = 32; SDO List.Disable PDO.AbortIfError = FALSE; SDO List.Disable PDO.JumpToLine = FALSE; SDO List.Disable PDO.Line = 0; SDO List.Set transmission type.Index = 16#1801; SDO List.Set transmission type.Subindex = 16#02; SDO List.Set transmission type.Value = 16#FF; SDO List.Set transmission type.Size = 8; SDO List.Set transmission type.AbortIfError = FALSE; SDO List.Set transmission type.JumpToLine = FALSE; SDO List.Set transmission type.Line = 0; SDO List.Set inhibit time.Index = 16#1801; SDO List.Set inhibit time.Subindex = 16#03; SDO List.Set inhibit time.Value = 16#001E; SDO List.Set inhibit time.Size = 16; SDO List.Set inhibit time.AbortIfError = FALSE; SDO List.Set inhibit time.JumpToLine = FALSE; SDO List.Set inhibit time.Line = 0; SDO List.Set event time.Index = 16#1801; SDO List.Set event time.Subindex = 16#05; SDO List.Set event time.Value = 16#03E8; SDO List.Set event time.Size = 16; SDO List.Set event time.AbortIfError = FALSE; SDO List.Set event time.JumpToLine = FALSE; SDO List.Set event time.Line = 0; SDO List.Clear pdo mapping.Index = 16#1A01; SDO List.Clear pdo mapping.Subindex = 16#00; SDO List.Clear pdo mapping.Value = 16#0; SDO List.Clear pdo mapping.Size = 8; SDO List.Clear pdo mapping.AbortIfError = FALSE; SDO List.Clear pdo mapping.JumpToLine = FALSE; SDO List.Clear pdo mapping.Line = 0;
              SDO List.Set Mapping.Index = 16#1A01; SDO List.Set Mapping.Subindex = 16#01; SDO List.Set Mapping.Value = 16#60410010; SDO List.Set Mapping.Size = 32; SDO List.Set Mapping.AbortIfError = FALSE; SDO List.Set Mapping.JumpToLine = FALSE; SDO List.Set Mapping.Line = 0; SDO List.Set Mapping.Index = 16#1A01; SDO List.Set Mapping.Subindex = 16#02; SDO List.Set Mapping.Value = 16#20020710; SDO List.Set Mapping.Size = 32; SDO List.Set Mapping.AbortIfError = FALSE; SDO List.Set Mapping.JumpToLine = FALSE; SDO List.Set Mapping.Line = 0; SDO List.Set Mapping.Index = 16#1A01; SDO List.Set Mapping.Subindex = 16#03; SDO List.Set Mapping.Value = 16#60440010; SDO List.Set Mapping.Size = 32; SDO List.Set Mapping.AbortIfError = FALSE; SDO List.Set Mapping.JumpToLine = FALSE; SDO List.Set Mapping.Line = 0; SDO List.Set Mapping.Index = 16#1A01; SDO List.Set Mapping.Subindex = 16#04; SDO List.Set Mapping.Value = 16#20160310; SDO List.Set Mapping.Size = 32; SDO List.Set Mapping.AbortIfError = FALSE; SDO List.Set Mapping.JumpToLine = FALSE; SDO List.Set Mapping.Line = 0; SDO List.Set number of pdos.Index = 16#1A01; SDO List.Set number of pdos.Subindex = 16#00; SDO List.Set number of pdos.Value = 16#04; SDO List.Set number of pdos.Size = 8; SDO List.Set number of pdos.AbortIfError = FALSE; SDO List.Set number of pdos.JumpToLine = FALSE; SDO List.Set number of pdos.Line = 0; SDO List.Set and enable COB-ID.Index = 16#1801; SDO List.Set and enable COB-ID.Subindex = 16#01; SDO List.Set and enable COB-ID.Value = 16#00000283; SDO List.Set and enable COB-ID.Size = 32; SDO List.Set and enable COB-ID.AbortIfError = FALSE;
              SDO List.Set and enable COB-ID.JumpToLine = FALSE; SDO List.Set and enable COB-ID.Line = 0; ConfigVersion = 50659584
            output altivar_2_Controlword : UINT  // Controlword
            output altivar_2_HMI_Frequency_ref : INT  // HMI Frequency ref.
            input  altivar_2_OL1R : UINT  // OL1R
            input  altivar_2_Statusword : UINT  // Statusword
            input  altivar_2_ETI_state_word : UINT  // ETI state word
            input  altivar_2_Control_Effort : INT  // Control Effort
            input  altivar_2_IL1R : UINT  // IL1R
  HMIGTO5310_5315 : HMIGTO5310/5315, Schneider Electric, order no. HMIGTO5310/5315, version 3.5.3.46
    HMI Application
    COM1
      SoMachine_Network_Manager1 : SoMachine-Network Manager, Schneider Electric, version 4.0.0.2
    COM2
      SoMachine_Network_Manager2 : SoMachine-Network Manager, Schneider Electric, version 4.0.0.2
    Ethernet
      SoMachine_Network_Manager3 : SoMachine-Network Manager, Schneider Electric, version 4.0.0.2
    USB
      SoMachine_Network_Manager4 : SoMachine-Network Manager, Schneider Electric, version 4.0.0.2
  6c0f7fb6-600b-4c93-9262-20cdc603757e
*)

// MyController/Application/GVL
VAR_GLOBAL
	// Вертикальное перемещение режущей рамки вверх
	ctrld_CuttingFrame_up: BOOL;
	// Вертикальное перемещение режущей рамки вниз
	ctrld_CuttingFrame_dn: BOOL;
	var_CuttingFrame_freq_up: INT := 333;
	var_CuttingFrame_freq_dn: INT := 444;
	// Горизонтальное перемешение режущей рамки вперёд
	ctrld_MovingFrame_fwd: BOOL;
	// Горизонтальное перемешение режущей рамки назад
	ctrld_MovingFrame_rev: BOOL;
	var_MovingFrame_freq_fwd: INT := 111;
	var_MovingFrame_freq_rev: INT := 222;
	// Привод тросового толкателя до резчика (удаление)
	var_BeforeCutter_far: BOOL;
	// Привод тросового толкателя до резчика (приближение)
	var_BeforeCutter_near: BOOL;
	var_BeforeCutter_freq_far: INT := 555;
	var_BeforeCutter_freq_near: INT := 666;
	// KM2; привод струны на срезание горбушки
	var_KL01: BOOL;
	// KM3; электродвигатель боковой подрезки
	var_KL02: BOOL;
	// KM4; электродвигатель боковой подрезки 2
	var_KL03: BOOL;
	// KM5; тормоз горизонтальной разки
	var_KL04: BOOL;
	// KM6; тормоз вертикальной резки
	var_KL05: BOOL;
	// KM7; электродвигатель мешалки шлама
	var_KL06: BOOL;
	// KM8; электродвигатель мешалки шлама
	var_KL07: BOOL;
	// KM9; электродвигатель маслостанции 11кВт
	var_KL08: BOOL;
	// KM10; электродвигатель маслостанции 11кВт
	var_KL09: BOOL;
	// KM11; электродвигатель маслостанции 3кВт
	var_KL10: BOOL;
	// KM12; электродвигатель тросового толкателя после резчика
	var_KL11: BOOL;
	// KM12; электродвигатель тросового толкателя после резчика (реверс)
	var_KL12: BOOL;
	// KM13; электродвигатель тросового толкателя обгонного пути
	var_KL13: BOOL;
	// KM13; электродвигатель тросового толкателя обгонного пути (реверс)
	var_KL14: BOOL;
	// Звуковой сигнал
	var_KL15: BOOL;
	// Аварийный стоп
	var_KL16: BOOL;
	// Z1_+ Маслостанция
	var_KL17: BOOL;
	// Z2_+ Маслостанция
	var_KL18: BOOL;
	// Z3_+ Маслостанция
	var_KL19: BOOL;
	// Z4_+ Маслостанция
	var_KL20: BOOL;
	// Z5_+ Маслостанция
	var_KL21: BOOL;
	// Z6_+ Маслостанция
	var_KL22: BOOL;
	// Z7_+ Маслостанция
	var_KL23: BOOL;
	// Z8_+ Маслостанция
	var_KL24: BOOL;
	// Z9_+ Опрокидыватель
	var_KL25: BOOL;
	// Z10_+ Опрокидыватель
	var_KL26: BOOL;
	// Z11_+ Опрокидыватель
	var_KL27: BOOL;
	// Z12_+ Опрокидыватель
	var_KL28: BOOL;
	// Z13_+ Опрокидыватель
	var_KL29: BOOL;
	// Z14_+ Опрокидыватель
	var_KL30: BOOL;
	// Z15_+ Опрокидыватель
	var_KL31: BOOL;
	// Z16_+ Опрокидыватель
	var_KL32: BOOL;
	// Z17_+ Опрокидыватель
	var_KL33: BOOL;
	// Z18_+ Опрокидыватель
	var_KL34: BOOL;
	// Z19_+ Опрокидыватель
	var_KL35: BOOL;
	// Z20_+ Опрокидыватель
	var_KL36: BOOL;
	// Z21A_+ Маслостанция
	var_KL37: BOOL;
	// Z22A_+ Маслостанция
	var_KL38: BOOL;
	// Z23_+ Маслостанция
	var_KL39: BOOL;
	// Z24_+ Маслостанция
	var_KL40: BOOL;
	// Z25_+ Горизонтальная резка
	var_KL41: BOOL;
	// Z26_+ Горизонтальная резка
	var_KL42: BOOL;
	// Z0A_+ Маслостанция
	var_KL43: BOOL;
	// Z0B_+ Маслостанция
	var_KL44: BOOL;
	// Z0C_+ Маслостанция
	var_KL45: BOOL;
	// Z21B_+ Маслостанция
	var_KL46: BOOL;
	// Z22B_+ Маслостанция
	var_KL47: BOOL;
	var_KL48: BOOL;
	var_KL49: BOOL;
	var_KL50: BOOL;
	var_KL51: BOOL;
	var_KL52: BOOL;
	var_KL53: BOOL;
	var_KL54: BOOL;
	var_KL55: BOOL;
	var_KL56: BOOL;
	var_KL57: BOOL;
	var_KL58: BOOL;
	var_KL59: BOOL;
	var_KL60: BOOL;
	var_KL61: BOOL;
	var_KL62: BOOL;
	var_KL63: BOOL;
	var_KL64: BOOL;
	// байт аварий
	wAlarm: BYTE := 11;
	// Основной бит аварий
	bGlobalAlarm: BOOL := False;
	Buzer_start: BOOL;
	// Выбор режима Ручной/Авто
	bGlobalAuto: BOOL;
	// для отладки (блокировка физических сигналов)
	bGlobalDebug: BOOL;
	// Блокировка действий на остальных этапах
	bGlobalLock: BOOL;
	wStep: INT;
END_VAR

// MyController/Application/POU_outputs_11_20
PROGRAM POU_outputs_11_20

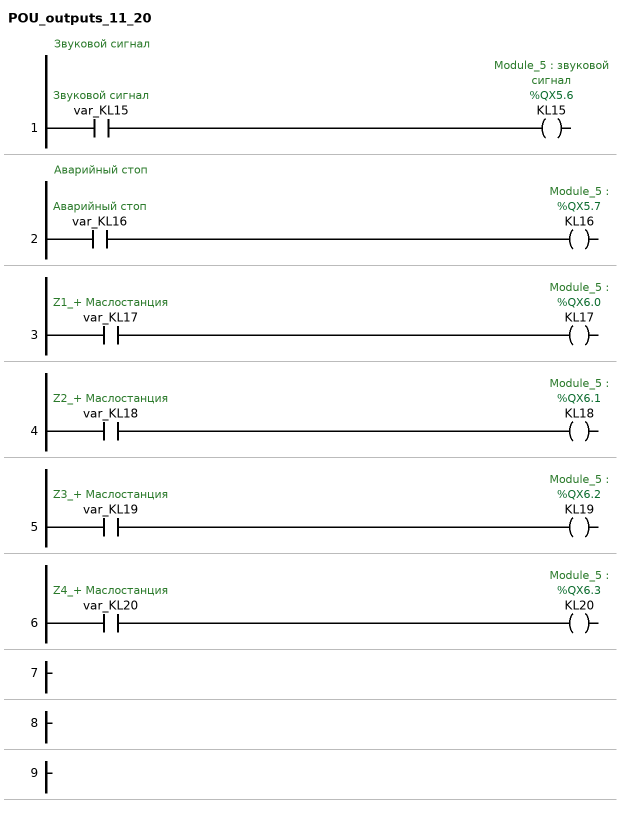
// NETWORK 1
// Звуковой сигнал
//   var_KL15: Звуковой сигнал
//   KL15: Module_5 : звуковой сигнал | AT %QX5.6
KL15 := var_KL15;

// NETWORK 2
// Аварийный стоп
//   var_KL16: Аварийный стоп
//   KL16: Module_5 : | AT %QX5.7
KL16 := var_KL16;

// NETWORK 3
//   var_KL17: Z1_+ Маслостанция
//   KL17: Module_5 : | AT %QX6.0
KL17 := var_KL17;

// NETWORK 4
//   var_KL18: Z2_+ Маслостанция
//   KL18: Module_5 : | AT %QX6.1
KL18 := var_KL18;

// NETWORK 5
//   var_KL19: Z3_+ Маслостанция
//   KL19: Module_5 : | AT %QX6.2
KL19 := var_KL19;

// NETWORK 6
//   var_KL20: Z4_+ Маслостанция
//   KL20: Module_5 : | AT %QX6.3
KL20 := var_KL20;

// NETWORK 7

// NETWORK 8

// NETWORK 9

END_PROGRAM

// MyController/Application/POU_outputs_21_30
PROGRAM POU_outputs_21_30

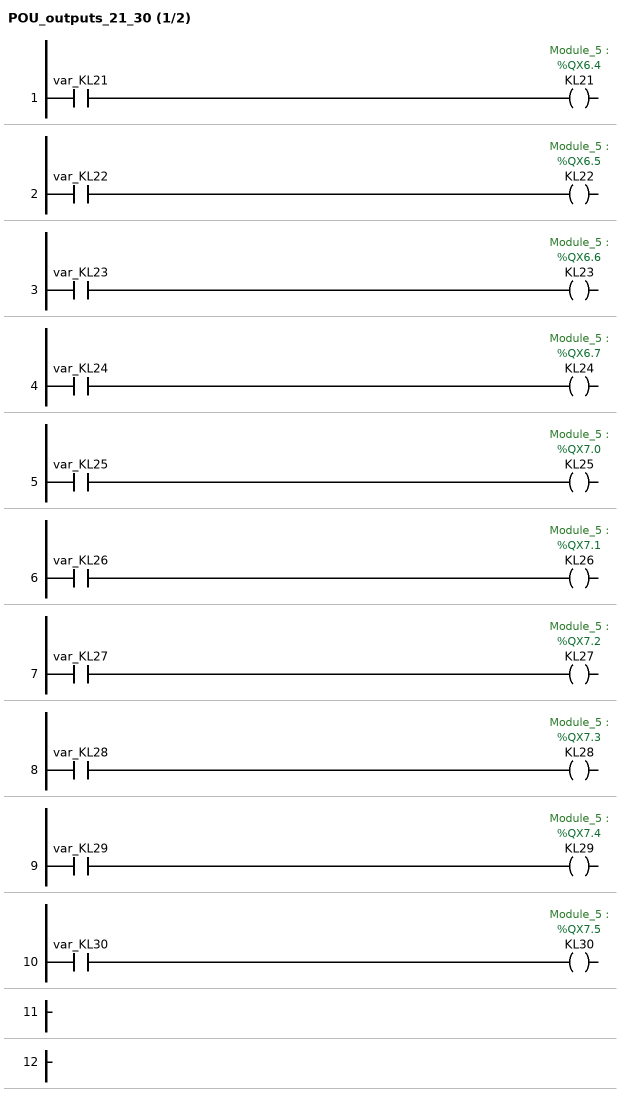
// NETWORK 1
//   KL21: Module_5 : | AT %QX6.4
KL21 := var_KL21;

// NETWORK 2
//   KL22: Module_5 : | AT %QX6.5
KL22 := var_KL22;

// NETWORK 3
//   KL23: Module_5 : | AT %QX6.6
KL23 := var_KL23;

// NETWORK 4
//   KL24: Module_5 : | AT %QX6.7
KL24 := var_KL24;

// NETWORK 5
//   KL25: Module_5 : | AT %QX7.0
KL25 := var_KL25;

// NETWORK 6
//   KL26: Module_5 : | AT %QX7.1
KL26 := var_KL26;

// NETWORK 7
//   KL27: Module_5 : | AT %QX7.2
KL27 := var_KL27;

// NETWORK 8
//   KL28: Module_5 : | AT %QX7.3
KL28 := var_KL28;

// NETWORK 9
//   KL29: Module_5 : | AT %QX7.4
KL29 := var_KL29;

// NETWORK 10
//   KL30: Module_5 : | AT %QX7.5
KL30 := var_KL30;

// NETWORK 11

// NETWORK 12

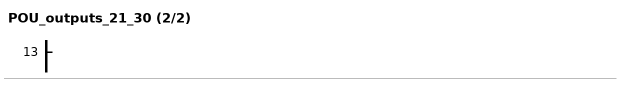
// NETWORK 13

END_PROGRAM

// MyController/Application/POU_outputs_31_40
PROGRAM POU_outputs_31_40

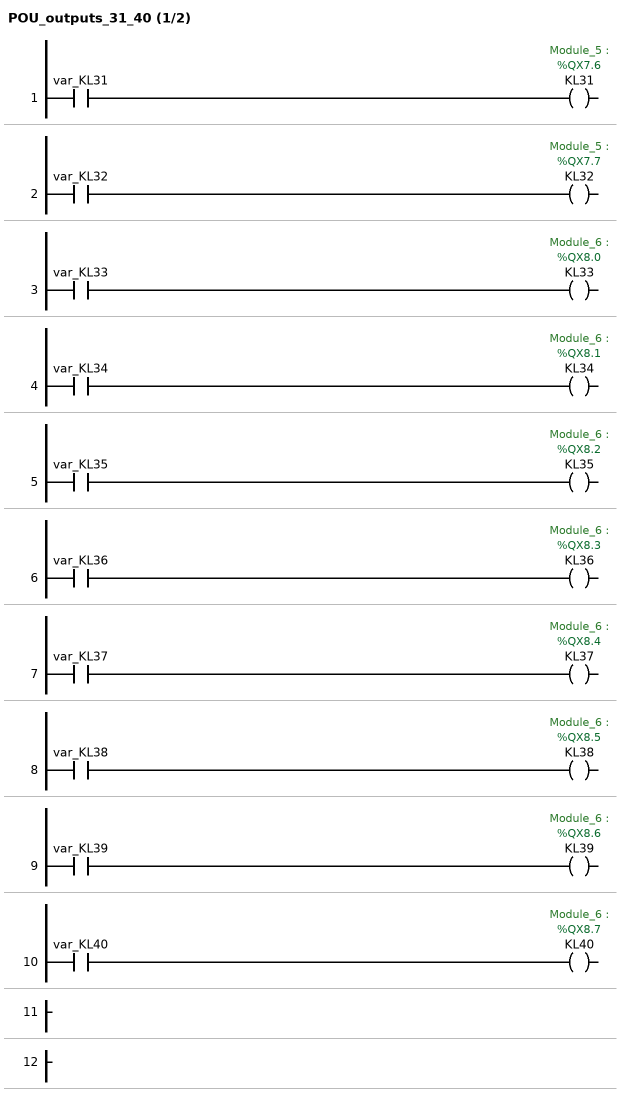
// NETWORK 1
//   KL31: Module_5 : | AT %QX7.6
KL31 := var_KL31;

// NETWORK 2
//   KL32: Module_5 : | AT %QX7.7
KL32 := var_KL32;

// NETWORK 3
//   KL33: Module_6 : | AT %QX8.0
KL33 := var_KL33;

// NETWORK 4
//   KL34: Module_6 : | AT %QX8.1
KL34 := var_KL34;

// NETWORK 5
//   KL35: Module_6 : | AT %QX8.2
KL35 := var_KL35;

// NETWORK 6
//   KL36: Module_6 : | AT %QX8.3
KL36 := var_KL36;

// NETWORK 7
//   KL37: Module_6 : | AT %QX8.4
KL37 := var_KL37;

// NETWORK 8
//   KL38: Module_6 : | AT %QX8.5
KL38 := var_KL38;

// NETWORK 9
//   KL39: Module_6 : | AT %QX8.6
KL39 := var_KL39;

// NETWORK 10
//   KL40: Module_6 : | AT %QX8.7
KL40 := var_KL40;

// NETWORK 11

// NETWORK 12

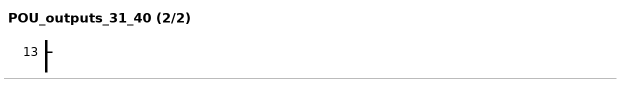
// NETWORK 13

END_PROGRAM

// MyController/Application/POU_outputs_41_50
PROGRAM POU_outputs_41_50

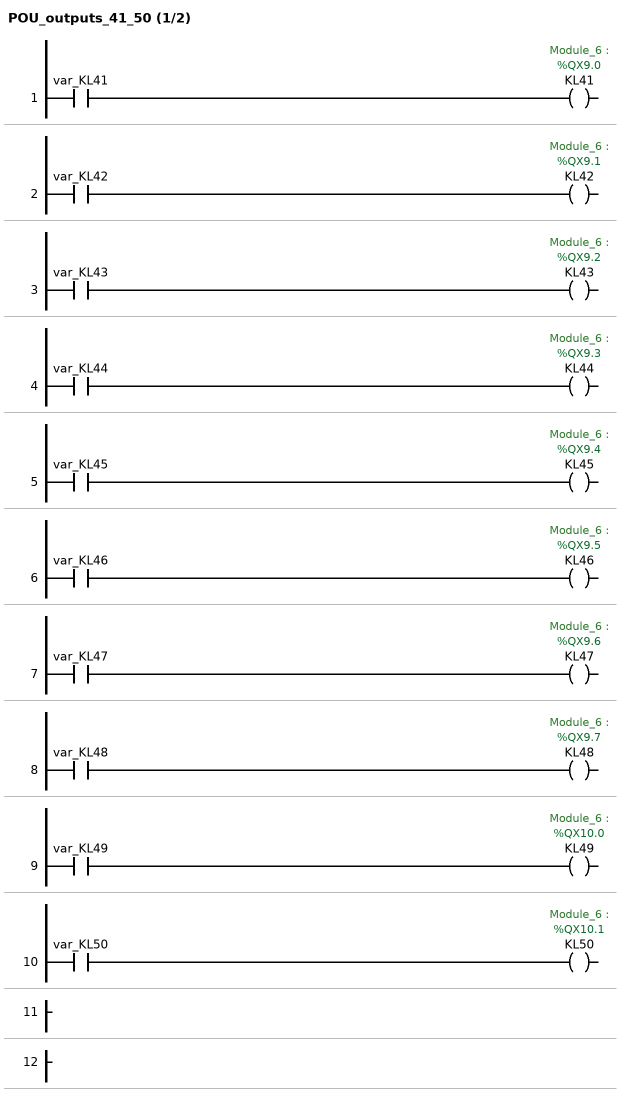
// NETWORK 1
//   KL41: Module_6 : | AT %QX9.0
KL41 := var_KL41;

// NETWORK 2
//   KL42: Module_6 : | AT %QX9.1
KL42 := var_KL42;

// NETWORK 3
//   KL43: Module_6 : | AT %QX9.2
KL43 := var_KL43;

// NETWORK 4
//   KL44: Module_6 : | AT %QX9.3
KL44 := var_KL44;

// NETWORK 5
//   KL45: Module_6 : | AT %QX9.4
KL45 := var_KL45;

// NETWORK 6
//   KL46: Module_6 : | AT %QX9.5
KL46 := var_KL46;

// NETWORK 7
//   KL47: Module_6 : | AT %QX9.6
KL47 := var_KL47;

// NETWORK 8
//   KL48: Module_6 : | AT %QX9.7
KL48 := var_KL48;

// NETWORK 9
//   KL49: Module_6 : | AT %QX10.0
KL49 := var_KL49;

// NETWORK 10
//   KL50: Module_6 : | AT %QX10.1
KL50 := var_KL50;

// NETWORK 11

// NETWORK 12

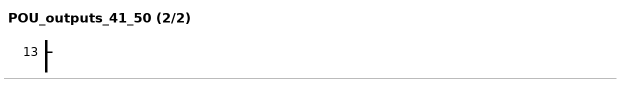
// NETWORK 13

END_PROGRAM

// MyController/Application/POU_outputs_51_64
PROGRAM POU_outputs_51_64

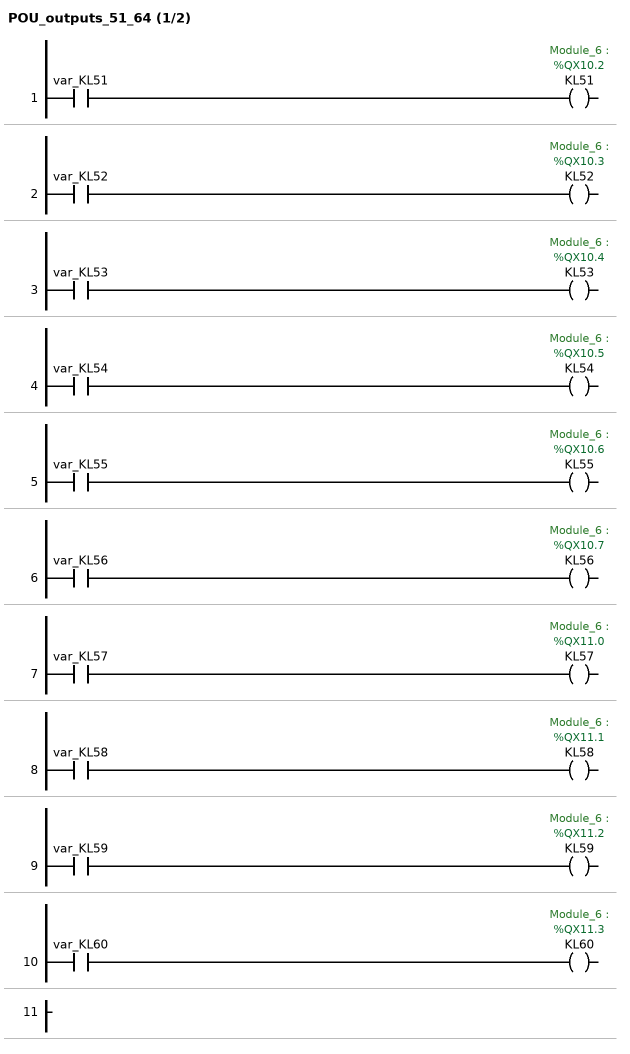
// NETWORK 1
//   KL51: Module_6 : | AT %QX10.2
KL51 := var_KL51;

// NETWORK 2
//   KL52: Module_6 : | AT %QX10.3
KL52 := var_KL52;

// NETWORK 3
//   KL53: Module_6 : | AT %QX10.4
KL53 := var_KL53;

// NETWORK 4
//   KL54: Module_6 : | AT %QX10.5
KL54 := var_KL54;

// NETWORK 5
//   KL55: Module_6 : | AT %QX10.6
KL55 := var_KL55;

// NETWORK 6
//   KL56: Module_6 : | AT %QX10.7
KL56 := var_KL56;

// NETWORK 7
//   KL57: Module_6 : | AT %QX11.0
KL57 := var_KL57;

// NETWORK 8
//   KL58: Module_6 : | AT %QX11.1
KL58 := var_KL58;

// NETWORK 9
//   KL59: Module_6 : | AT %QX11.2
KL59 := var_KL59;

// NETWORK 10
//   KL60: Module_6 : | AT %QX11.3
KL60 := var_KL60;

// NETWORK 11

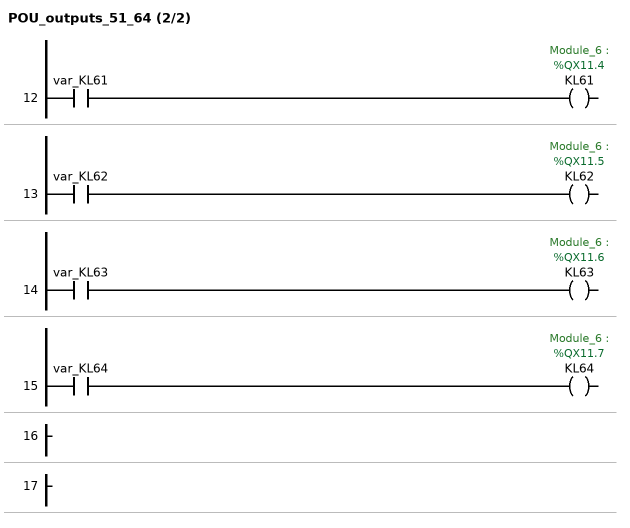
// NETWORK 12
//   KL61: Module_6 : | AT %QX11.4
KL61 := var_KL61;

// NETWORK 13
//   KL62: Module_6 : | AT %QX11.5
KL62 := var_KL62;

// NETWORK 14
//   KL63: Module_6 : | AT %QX11.6
KL63 := var_KL63;

// NETWORK 15
//   KL64: Module_6 : | AT %QX11.7
KL64 := var_KL64;

// NETWORK 16

// NETWORK 17

END_PROGRAM

// MyController/Application/POU_outputs_drivers
PROGRAM POU_outputs_drivers

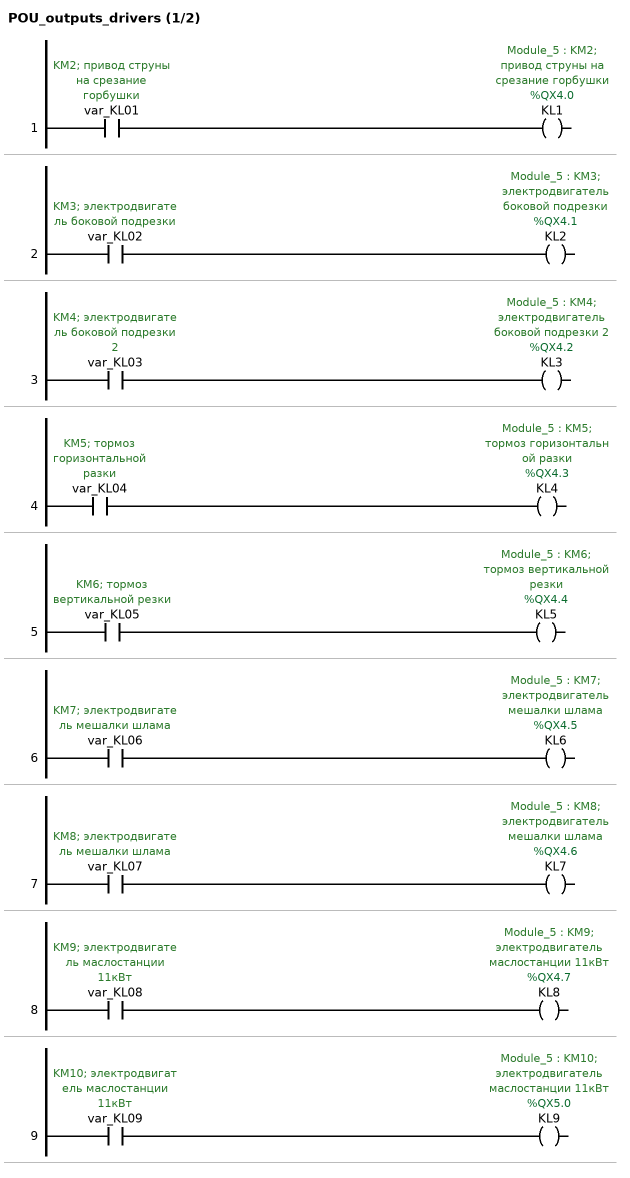
// NETWORK 1
//   var_KL01: KM2; привод струны на срезание горбушки
//   KL1: Module_5 : KM2; привод струны на срезание горбушки | AT %QX4.0
KL1 := var_KL01;

// NETWORK 2
//   var_KL02: KM3; электродвигатель боковой подрезки
//   KL2: Module_5 : KM3; электродвигатель боковой подрезки | AT %QX4.1
KL2 := var_KL02;

// NETWORK 3
//   var_KL03: KM4; электродвигатель боковой подрезки 2
//   KL3: Module_5 : KM4; электродвигатель боковой подрезки 2 | AT %QX4.2
KL3 := var_KL03;

// NETWORK 4
//   var_KL04: KM5; тормоз горизонтальной разки
//   KL4: Module_5 : KM5; тормоз горизонтальной разки | AT %QX4.3
KL4 := var_KL04;

// NETWORK 5
//   var_KL05: KM6; тормоз вертикальной резки
//   KL5: Module_5 : KM6; тормоз вертикальной резки | AT %QX4.4
KL5 := var_KL05;

// NETWORK 6
//   var_KL06: KM7; электродвигатель мешалки шлама
//   KL6: Module_5 : KM7; электродвигатель мешалки шлама | AT %QX4.5
KL6 := var_KL06;

// NETWORK 7
//   var_KL07: KM8; электродвигатель мешалки шлама
//   KL7: Module_5 : KM8; электродвигатель мешалки шлама | AT %QX4.6
KL7 := var_KL07;

// NETWORK 8
//   var_KL08: KM9; электродвигатель маслостанции 11кВт
//   KL8: Module_5 : KM9; электродвигатель маслостанции 11кВт | AT %QX4.7
KL8 := var_KL08;

// NETWORK 9
//   var_KL09: KM10; электродвигатель маслостанции 11кВт
//   KL9: Module_5 : KM10; электродвигатель маслостанции 11кВт | AT %QX5.0
KL9 := var_KL09;

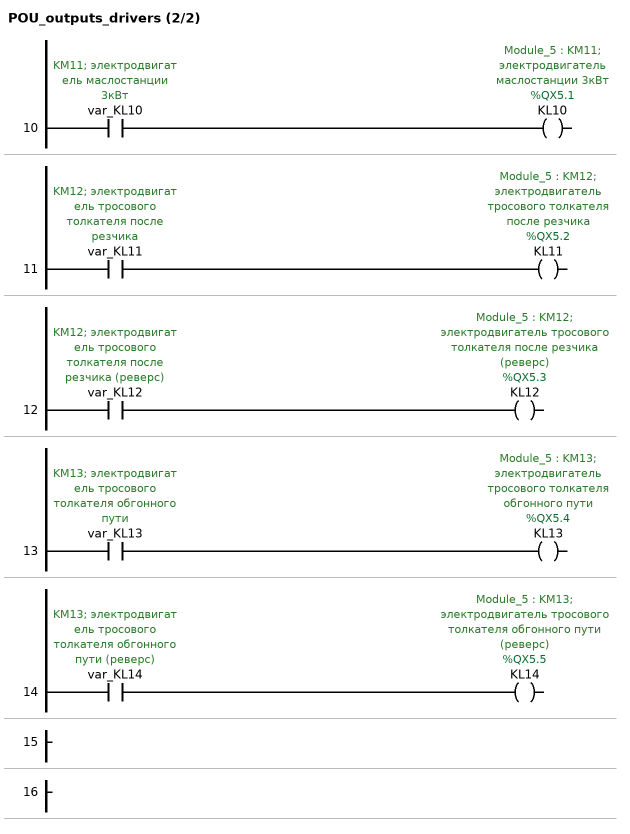
// NETWORK 10
//   var_KL10: KM11; электродвигатель маслостанции 3кВт
//   KL10: Module_5 : KM11; электродвигатель маслостанции 3кВт | AT %QX5.1
KL10 := var_KL10;

// NETWORK 11
//   var_KL11: KM12; электродвигатель тросового толкателя после резчика
//   KL11: Module_5 : KM12; электродвигатель тросового толкателя после резчика | AT %QX5.2
KL11 := var_KL11;

// NETWORK 12
//   var_KL12: KM12; электродвигатель тросового толкателя после резчика (реверс)
//   KL12: Module_5 : KM12; электродвигатель тросового толкателя после резчика (реверс) | AT %QX5.3
KL12 := var_KL12;

// NETWORK 13
//   var_KL13: KM13; электродвигатель тросового толкателя обгонного пути
//   KL13: Module_5 : KM13; электродвигатель тросового толкателя обгонного пути | AT %QX5.4
KL13 := var_KL13;

// NETWORK 14
//   var_KL14: KM13; электродвигатель тросового толкателя обгонного пути (реверс)
//   KL14: Module_5 : KM13; электродвигатель тросового толкателя обгонного пути (реверс) | AT %QX5.5
KL14 := var_KL14;

// NETWORK 15

// NETWORK 16

END_PROGRAM

// MyController/Application/POU_10_outputs_oilstation
PROGRAM POU_10_outputs_oilstation

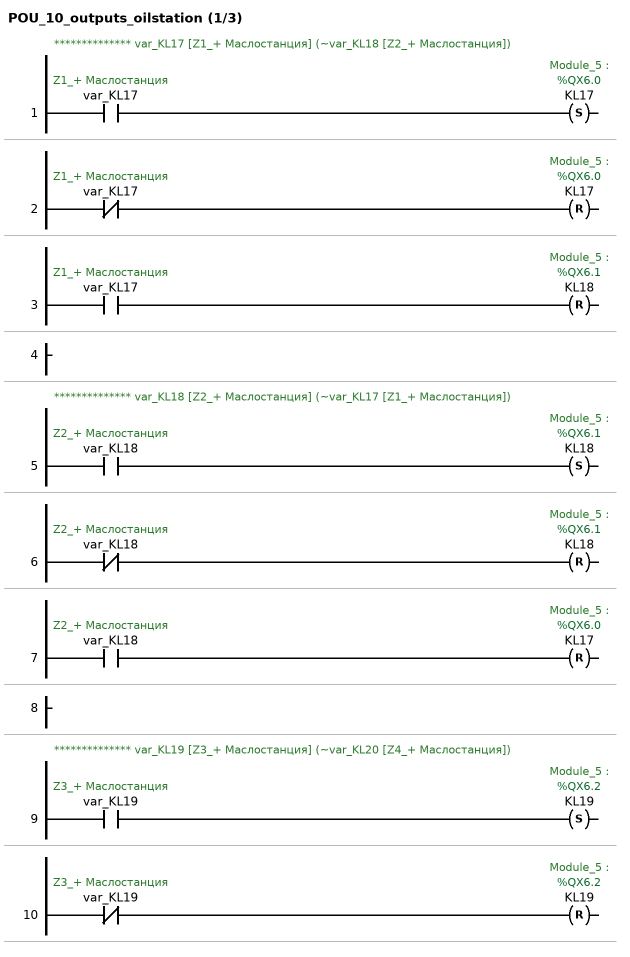
// NETWORK 1
// ************** var_KL17 [Z1_+ Маслостанция] (~var_KL18 [Z2_+ Маслостанция])
//   var_KL17: Z1_+ Маслостанция
//   KL17: Module_5 : | AT %QX6.0
KL17 S= var_KL17;

// NETWORK 2
//   var_KL17: Z1_+ Маслостанция
//   KL17: Module_5 : | AT %QX6.0
KL17 R= NOT var_KL17;

// NETWORK 3
//   var_KL17: Z1_+ Маслостанция
//   KL18: Module_5 : | AT %QX6.1
KL18 R= var_KL17;

// NETWORK 4

// NETWORK 5
// ************** var_KL18 [Z2_+ Маслостанция] (~var_KL17 [Z1_+ Маслостанция])
//   var_KL18: Z2_+ Маслостанция
//   KL18: Module_5 : | AT %QX6.1
KL18 S= var_KL18;

// NETWORK 6
//   var_KL18: Z2_+ Маслостанция
//   KL18: Module_5 : | AT %QX6.1
KL18 R= NOT var_KL18;

// NETWORK 7
//   var_KL18: Z2_+ Маслостанция
//   KL17: Module_5 : | AT %QX6.0
KL17 R= var_KL18;

// NETWORK 8

// NETWORK 9
// ************** var_KL19 [Z3_+ Маслостанция] (~var_KL20 [Z4_+ Маслостанция])
//   var_KL19: Z3_+ Маслостанция
//   KL19: Module_5 : | AT %QX6.2
KL19 S= var_KL19;

// NETWORK 10
//   var_KL19: Z3_+ Маслостанция
//   KL19: Module_5 : | AT %QX6.2
KL19 R= NOT var_KL19;

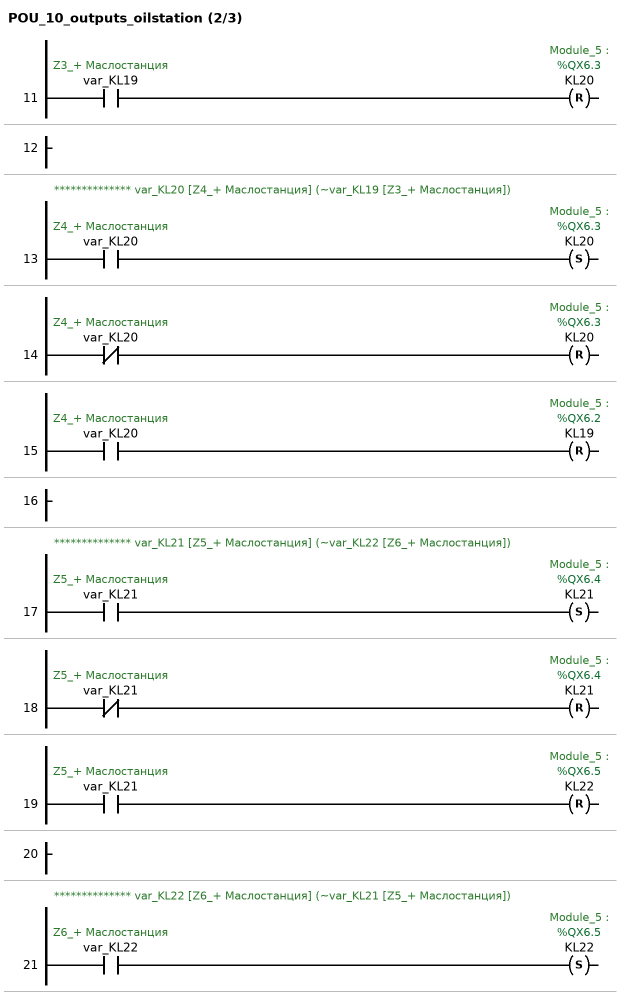
// NETWORK 11
//   var_KL19: Z3_+ Маслостанция
//   KL20: Module_5 : | AT %QX6.3
KL20 R= var_KL19;

// NETWORK 12

// NETWORK 13
// ************** var_KL20 [Z4_+ Маслостанция] (~var_KL19 [Z3_+ Маслостанция])
//   var_KL20: Z4_+ Маслостанция
//   KL20: Module_5 : | AT %QX6.3
KL20 S= var_KL20;

// NETWORK 14
//   var_KL20: Z4_+ Маслостанция
//   KL20: Module_5 : | AT %QX6.3
KL20 R= NOT var_KL20;

// NETWORK 15
//   var_KL20: Z4_+ Маслостанция
//   KL19: Module_5 : | AT %QX6.2
KL19 R= var_KL20;

// NETWORK 16

// NETWORK 17
// ************** var_KL21 [Z5_+ Маслостанция] (~var_KL22 [Z6_+ Маслостанция])
//   var_KL21: Z5_+ Маслостанция
//   KL21: Module_5 : | AT %QX6.4
KL21 S= var_KL21;

// NETWORK 18
//   var_KL21: Z5_+ Маслостанция
//   KL21: Module_5 : | AT %QX6.4
KL21 R= NOT var_KL21;

// NETWORK 19
//   var_KL21: Z5_+ Маслостанция
//   KL22: Module_5 : | AT %QX6.5
KL22 R= var_KL21;

// NETWORK 20

// NETWORK 21
// ************** var_KL22 [Z6_+ Маслостанция] (~var_KL21 [Z5_+ Маслостанция])
//   var_KL22: Z6_+ Маслостанция
//   KL22: Module_5 : | AT %QX6.5
KL22 S= var_KL22;

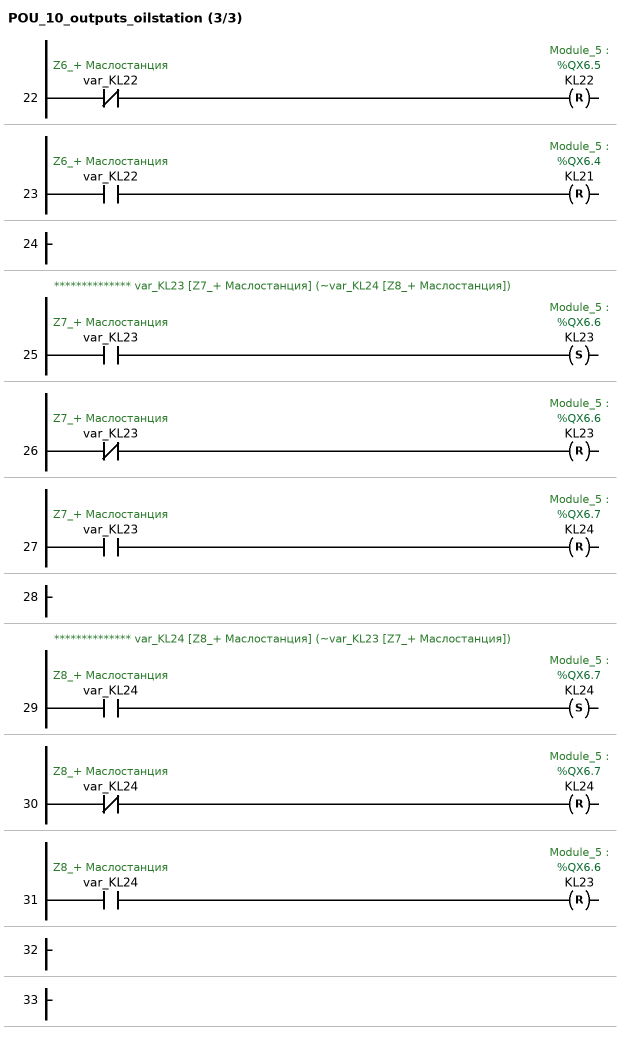
// NETWORK 22
//   var_KL22: Z6_+ Маслостанция
//   KL22: Module_5 : | AT %QX6.5
KL22 R= NOT var_KL22;

// NETWORK 23
//   var_KL22: Z6_+ Маслостанция
//   KL21: Module_5 : | AT %QX6.4
KL21 R= var_KL22;

// NETWORK 24

// NETWORK 25
// ************** var_KL23 [Z7_+ Маслостанция] (~var_KL24 [Z8_+ Маслостанция])
//   var_KL23: Z7_+ Маслостанция
//   KL23: Module_5 : | AT %QX6.6
KL23 S= var_KL23;

// NETWORK 26
//   var_KL23: Z7_+ Маслостанция
//   KL23: Module_5 : | AT %QX6.6
KL23 R= NOT var_KL23;

// NETWORK 27
//   var_KL23: Z7_+ Маслостанция
//   KL24: Module_5 : | AT %QX6.7
KL24 R= var_KL23;

// NETWORK 28

// NETWORK 29
// ************** var_KL24 [Z8_+ Маслостанция] (~var_KL23 [Z7_+ Маслостанция])
//   var_KL24: Z8_+ Маслостанция
//   KL24: Module_5 : | AT %QX6.7
KL24 S= var_KL24;

// NETWORK 30
//   var_KL24: Z8_+ Маслостанция
//   KL24: Module_5 : | AT %QX6.7
KL24 R= NOT var_KL24;

// NETWORK 31
//   var_KL24: Z8_+ Маслостанция
//   KL23: Module_5 : | AT %QX6.6
KL23 R= var_KL24;

// NETWORK 32

// NETWORK 33

END_PROGRAM

// MyController/Application/POU_1_Utils
PROGRAM POU_1_Utils
VAR
	sum: WORD;
	CTU_out: BOOL;
	CTU_0: CTU;
	BLINK_0: BLINK;
END_VAR
VAR // added by the converter: edge detectors and wires of the graphical bodies
    _ft1 : F_TRIG;
END_VAR

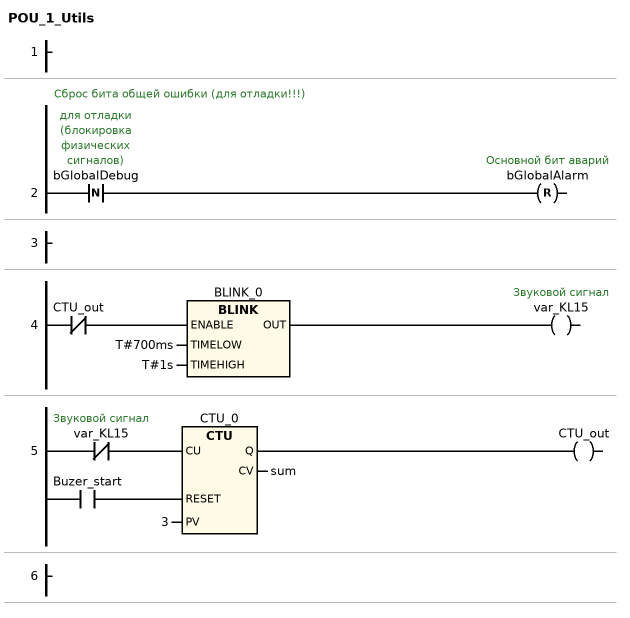
// NETWORK 1

// NETWORK 2
// Сброс бита общей ошибки (для отладки!!!)
//   bGlobalDebug: для отладки (блокировка физических сигналов)
//   bGlobalAlarm: Основной бит аварий
_ft1(CLK := bGlobalDebug);
bGlobalAlarm R= _ft1.Q;

// NETWORK 3

// NETWORK 4
//   var_KL15: Звуковой сигнал
BLINK_0(ENABLE := NOT CTU_out, TIMELOW := T#700ms, TIMEHIGH := T#1s); // BLINK
var_KL15 := BLINK_0.OUT;

// NETWORK 5
//   var_KL15: Звуковой сигнал
CTU_0(CU := NOT var_KL15, RESET := Buzer_start, PV := 3, CV => sum); // CTU
CTU_out := CTU_0.Q;

// NETWORK 6

END_PROGRAM

// MyController/Application/POU_2_TrosTolkateli
PROGRAM POU_2_TrosTolkateli

VAR
	lim_BeforeCutter_far: BOOL;
	lim_BeforeCutter_near: BOOL;
	post_BeforeCutter_far: BOOL;
	post_BeforeCutter_near: BOOL;
	ctrl_BeforeCutter_near: BOOL;
	// для управления приводом в автоматическом режиме
	ctrl_BeforeCutter_far: BOOL;
	sum_BeforeCutter_far: BOOL;
	sum_BeforeCutter_near: BOOL;
	// сигнал управления приводами
	drv_ctrl_BeforeCutter_far: BOOL;
	// Сигнал управления приводами
	drv_ctrl_BeforeCutter_near: BOOL;
	lim_AfterCutter_far: BOOL;
	lim_AfterCutter_near: BOOL;
	post_AfterCutter_far: BOOL;
	post_AfterCutter_near: BOOL;
	ctrl_AfterCutter_far: BOOL;
	ctrl_AfterCutter_near: BOOL;
	sum_ctrl_AfterCutter_far: BOOL;
	sum_ctrl_AfterCutter_near: BOOL;
	drv_ctrl_AfterCutter_near: BOOL;
	drv_ctrl_AfterCutter_far: BOOL;
	ctrl_BackPath_far: BOOL;
	ctrl_BackPath_near: BOOL;
	sum_ctrl_BackPath_far: BOOL;
	sum_ctrl_BackPath_near: BOOL;
	lim_BackPath_far: BOOL;
	lim_BackPath_near: BOOL;
	drv_ctrl_BackPath_far: BOOL;
	drv_ctrl_BackPath_near: BOOL;
END_VAR
VAR // added by the converter: edge detectors and wires of the graphical bodies
    _w1, _w2, _w3, _w4 : BOOL;
END_VAR

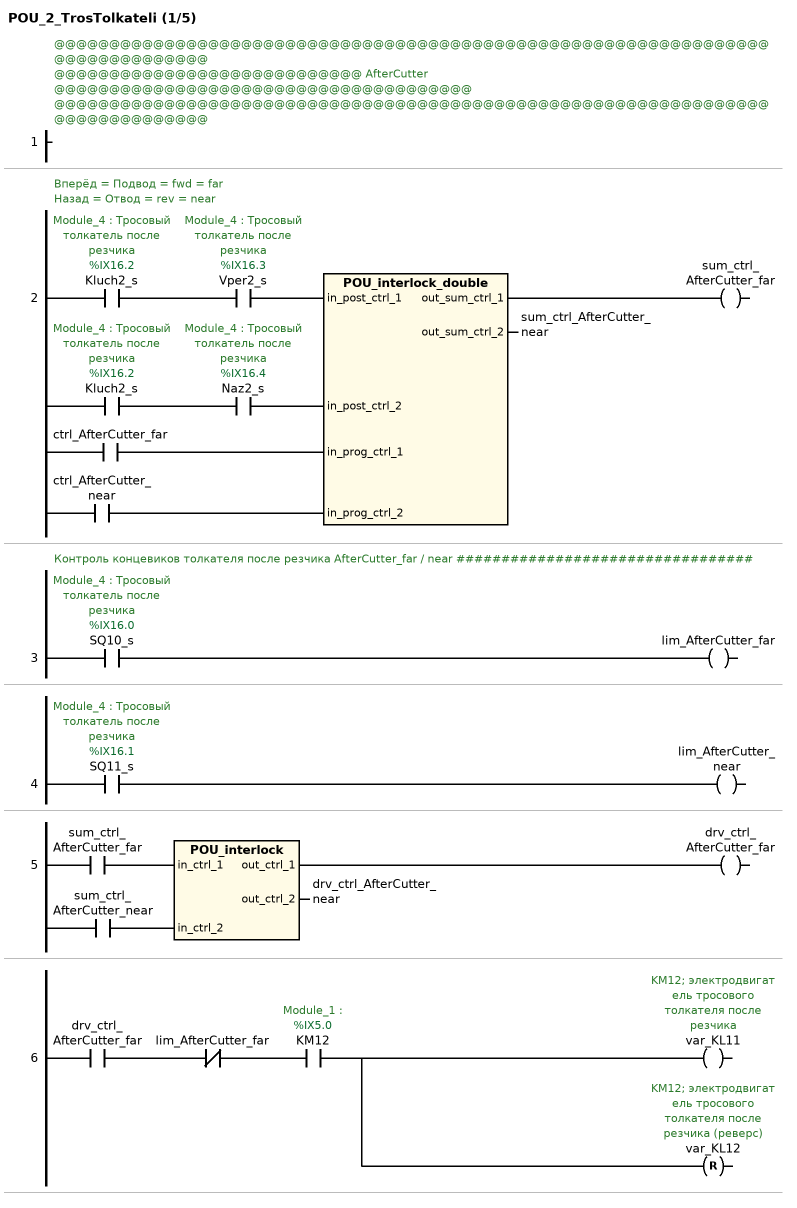
// NETWORK 1
// @@@@@@@@@@@@@@@@@@@@@@@@@@@@@@@@@@@@@@@@@@@@@@@@@@@@@@@@@@@@@@@@@@@@@@@@@@@@@@@
// @@@@@@@@@@@@@@@@@@@@@@@@@@@@ AfterCutter @@@@@@@@@@@@@@@@@@@@@@@@@@@@@@@@@@@@@@
// @@@@@@@@@@@@@@@@@@@@@@@@@@@@@@@@@@@@@@@@@@@@@@@@@@@@@@@@@@@@@@@@@@@@@@@@@@@@@@@

// NETWORK 2
// Вперёд = Подвод = fwd = far
// Назад = Отвод = rev = near
//   Kluch2_s: Module_4 : Тросовый толкатель после резчика | AT %IX16.2
//   Vper2_s: Module_4 : Тросовый толкатель после резчика | AT %IX16.3
//   Naz2_s: Module_4 : Тросовый толкатель после резчика | AT %IX16.4
POU_interlock_double(in_post_ctrl_1 := Kluch2_s AND Vper2_s, in_post_ctrl_2 := Kluch2_s AND Naz2_s, in_prog_ctrl_1 := ctrl_AfterCutter_far, in_prog_ctrl_2 := ctrl_AfterCutter_near, out_sum_ctrl_2 => sum_ctrl_AfterCutter_near);
sum_ctrl_AfterCutter_far := POU_interlock_double.out_sum_ctrl_1;

// NETWORK 3
// Контроль концевиков толкателя после резчика AfterCutter_far / near #################################
//   SQ10_s: Module_4 : Тросовый толкатель после резчика | AT %IX16.0
lim_AfterCutter_far := SQ10_s;

// NETWORK 4
//   SQ11_s: Module_4 : Тросовый толкатель после резчика | AT %IX16.1
lim_AfterCutter_near := SQ11_s;

// NETWORK 5
POU_interlock(in_ctrl_1 := sum_ctrl_AfterCutter_far, in_ctrl_2 := sum_ctrl_AfterCutter_near, out_ctrl_2 => drv_ctrl_AfterCutter_near);
drv_ctrl_AfterCutter_far := POU_interlock.out_ctrl_1;

// NETWORK 6
//   KM12: Module_1 : | AT %IX5.0
//   var_KL11: KM12; электродвигатель тросового толкателя после резчика
//   var_KL12: KM12; электродвигатель тросового толкателя после резчика (реверс)
_w1 := drv_ctrl_AfterCutter_far AND NOT lim_AfterCutter_far AND KM12;
var_KL11 := _w1;
var_KL12 R= _w1;

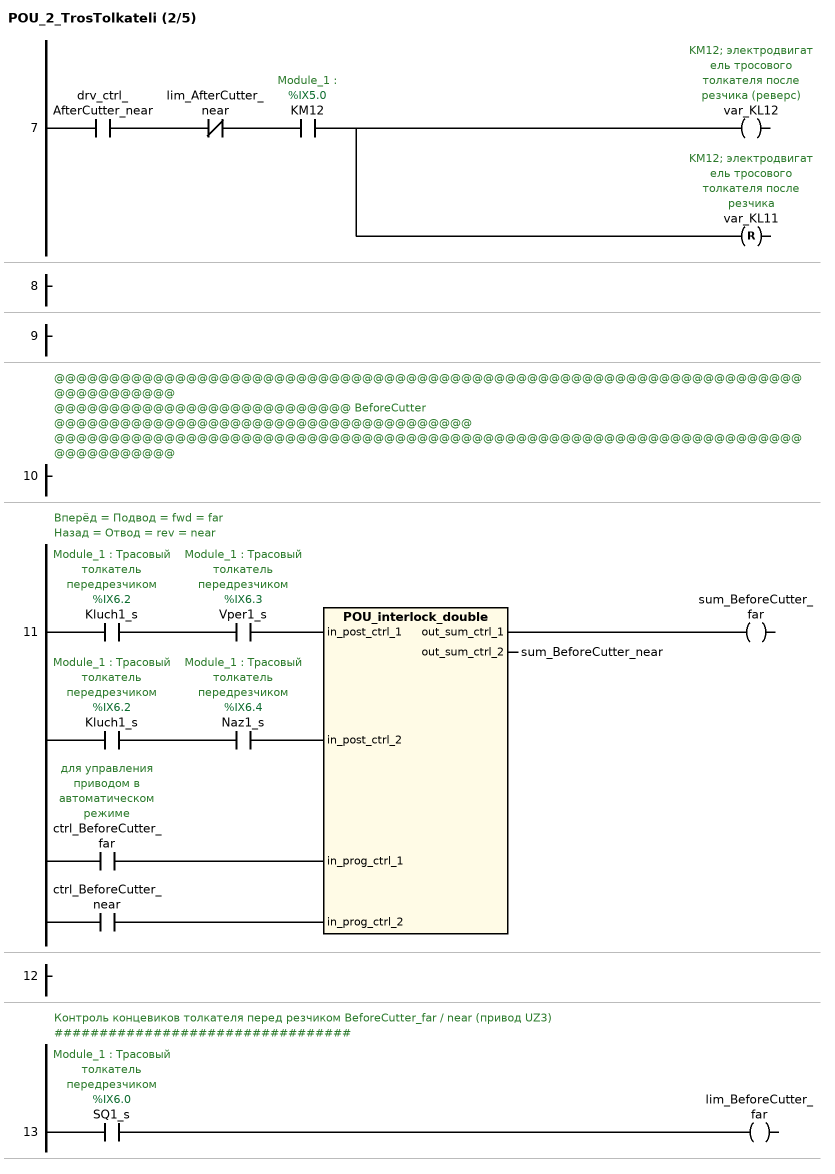
// NETWORK 7
//   KM12: Module_1 : | AT %IX5.0
//   var_KL12: KM12; электродвигатель тросового толкателя после резчика (реверс)
//   var_KL11: KM12; электродвигатель тросового толкателя после резчика
_w2 := drv_ctrl_AfterCutter_near AND NOT lim_AfterCutter_near AND KM12;
var_KL12 := _w2;
var_KL11 R= _w2;

// NETWORK 8

// NETWORK 9

// NETWORK 10
// @@@@@@@@@@@@@@@@@@@@@@@@@@@@@@@@@@@@@@@@@@@@@@@@@@@@@@@@@@@@@@@@@@@@@@@@@@@@@@@
// @@@@@@@@@@@@@@@@@@@@@@@@@@@ BeforeCutter @@@@@@@@@@@@@@@@@@@@@@@@@@@@@@@@@@@@@@
// @@@@@@@@@@@@@@@@@@@@@@@@@@@@@@@@@@@@@@@@@@@@@@@@@@@@@@@@@@@@@@@@@@@@@@@@@@@@@@@

// NETWORK 11
// Вперёд = Подвод = fwd = far
// Назад = Отвод = rev = near
//   Kluch1_s: Module_1 : Трасовый толкатель передрезчиком | AT %IX6.2
//   Vper1_s: Module_1 : Трасовый толкатель передрезчиком | AT %IX6.3
//   Naz1_s: Module_1 : Трасовый толкатель передрезчиком | AT %IX6.4
//   ctrl_BeforeCutter_far: для управления приводом в автоматическом режиме
POU_interlock_double(in_post_ctrl_1 := Kluch1_s AND Vper1_s, in_post_ctrl_2 := Kluch1_s AND Naz1_s, in_prog_ctrl_1 := ctrl_BeforeCutter_far, in_prog_ctrl_2 := ctrl_BeforeCutter_near, out_sum_ctrl_2 => sum_BeforeCutter_near);
sum_BeforeCutter_far := POU_interlock_double.out_sum_ctrl_1;

// NETWORK 12

// NETWORK 13
// Контроль концевиков толкателя перед резчиком BeforeCutter_far / near (привод UZ3) #################################
//   SQ1_s: Module_1 : Трасовый толкатель передрезчиком | AT %IX6.0
lim_BeforeCutter_far := SQ1_s;

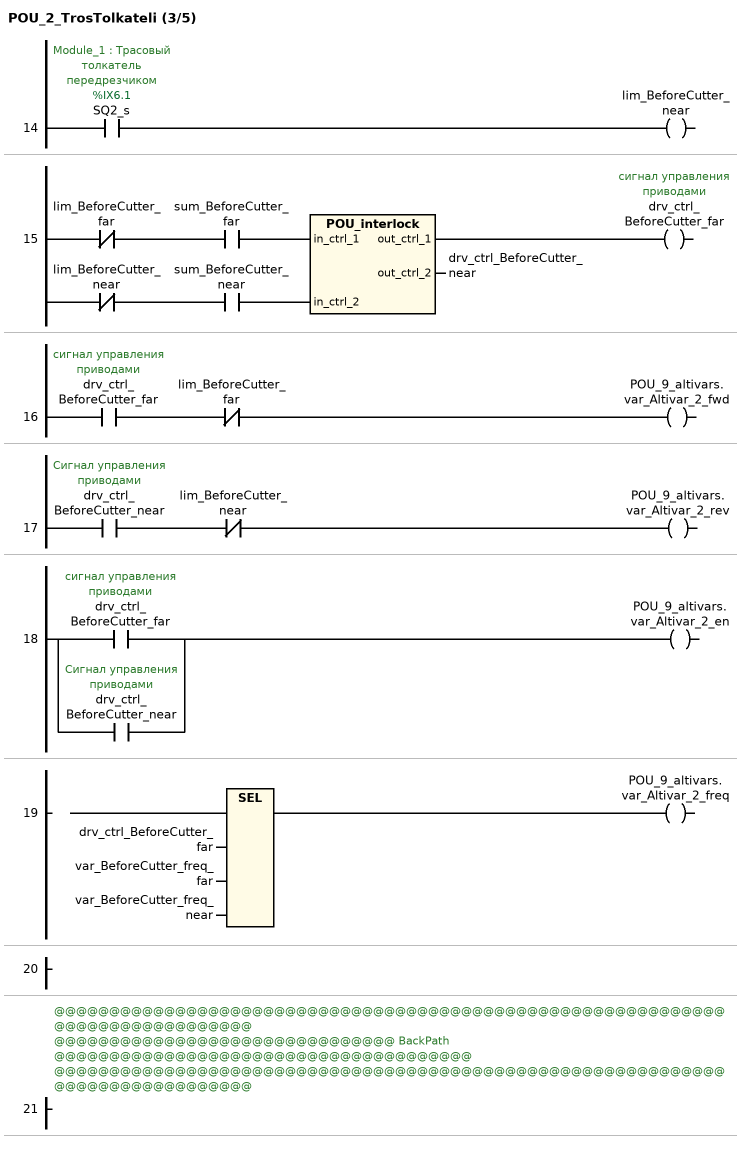
// NETWORK 14
//   SQ2_s: Module_1 : Трасовый толкатель передрезчиком | AT %IX6.1
lim_BeforeCutter_near := SQ2_s;

// NETWORK 15
//   drv_ctrl_BeforeCutter_near: Сигнал управления приводами
//   drv_ctrl_BeforeCutter_far: сигнал управления приводами
POU_interlock(in_ctrl_1 := NOT lim_BeforeCutter_far AND sum_BeforeCutter_far, in_ctrl_2 := NOT lim_BeforeCutter_near AND sum_BeforeCutter_near, out_ctrl_2 => drv_ctrl_BeforeCutter_near);
drv_ctrl_BeforeCutter_far := POU_interlock.out_ctrl_1;

// NETWORK 16
//   drv_ctrl_BeforeCutter_far: сигнал управления приводами
POU_9_altivars.var_Altivar_2_fwd := drv_ctrl_BeforeCutter_far AND NOT lim_BeforeCutter_far;

// NETWORK 17
//   drv_ctrl_BeforeCutter_near: Сигнал управления приводами
POU_9_altivars.var_Altivar_2_rev := drv_ctrl_BeforeCutter_near AND NOT lim_BeforeCutter_near;

// NETWORK 18
//   drv_ctrl_BeforeCutter_far: сигнал управления приводами
//   drv_ctrl_BeforeCutter_near: Сигнал управления приводами
POU_9_altivars.var_Altivar_2_en := drv_ctrl_BeforeCutter_far OR drv_ctrl_BeforeCutter_near;

// NETWORK 19
//   drv_ctrl_BeforeCutter_far: сигнал управления приводами
POU_9_altivars.var_Altivar_2_freq := SEL(drv_ctrl_BeforeCutter_far, var_BeforeCutter_freq_far, var_BeforeCutter_freq_near);

// NETWORK 20

// NETWORK 21
// @@@@@@@@@@@@@@@@@@@@@@@@@@@@@@@@@@@@@@@@@@@@@@@@@@@@@@@@@@@@@@@@@@@@@@@@@@@@@@@
// @@@@@@@@@@@@@@@@@@@@@@@@@@@@@@@ BackPath @@@@@@@@@@@@@@@@@@@@@@@@@@@@@@@@@@@@@@
// @@@@@@@@@@@@@@@@@@@@@@@@@@@@@@@@@@@@@@@@@@@@@@@@@@@@@@@@@@@@@@@@@@@@@@@@@@@@@@@

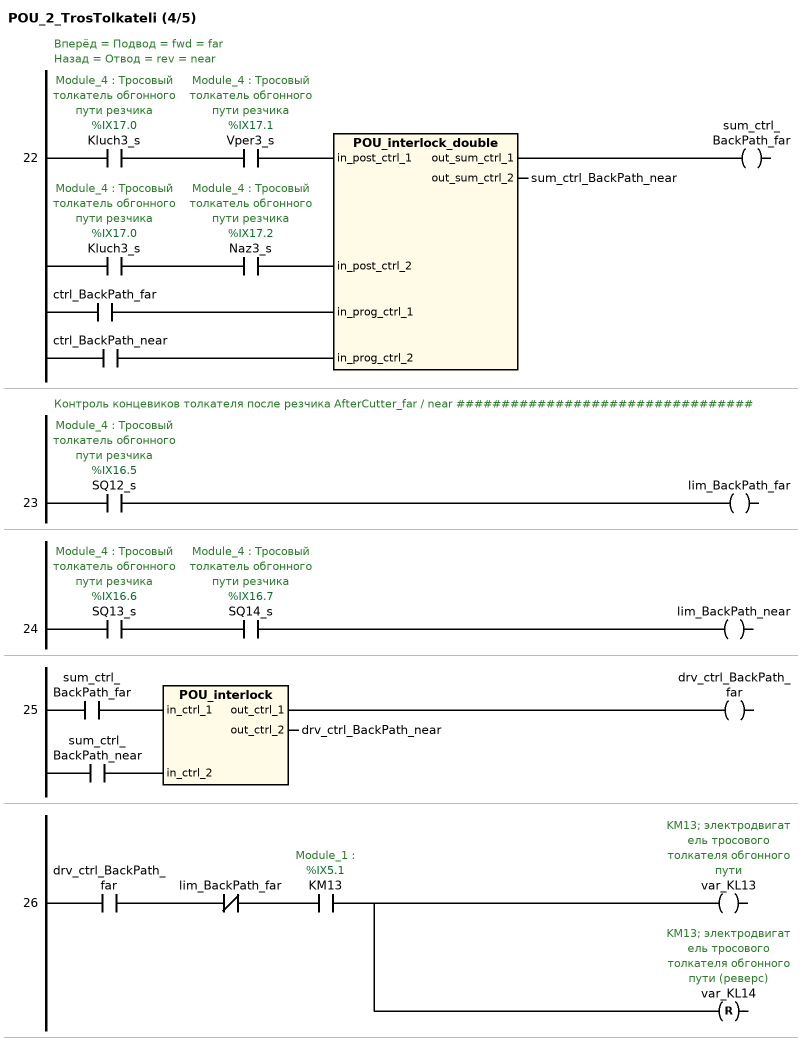
// NETWORK 22
// Вперёд = Подвод = fwd = far
// Назад = Отвод = rev = near
//   Kluch3_s: Module_4 : Тросовый толкатель обгонного пути резчика | AT %IX17.0
//   Vper3_s: Module_4 : Тросовый толкатель обгонного пути резчика | AT %IX17.1
//   Naz3_s: Module_4 : Тросовый толкатель обгонного пути резчика | AT %IX17.2
POU_interlock_double(in_post_ctrl_1 := Kluch3_s AND Vper3_s, in_post_ctrl_2 := Kluch3_s AND Naz3_s, in_prog_ctrl_1 := ctrl_BackPath_far, in_prog_ctrl_2 := ctrl_BackPath_near, out_sum_ctrl_2 => sum_ctrl_BackPath_near);
sum_ctrl_BackPath_far := POU_interlock_double.out_sum_ctrl_1;

// NETWORK 23
// Контроль концевиков толкателя после резчика AfterCutter_far / near #################################
//   SQ12_s: Module_4 : Тросовый толкатель обгонного пути резчика | AT %IX16.5
lim_BackPath_far := SQ12_s;

// NETWORK 24
//   SQ13_s: Module_4 : Тросовый толкатель обгонного пути резчика | AT %IX16.6
//   SQ14_s: Module_4 : Тросовый толкатель обгонного пути резчика | AT %IX16.7
lim_BackPath_near := SQ13_s AND SQ14_s;

// NETWORK 25
POU_interlock(in_ctrl_1 := sum_ctrl_BackPath_far, in_ctrl_2 := sum_ctrl_BackPath_near, out_ctrl_2 => drv_ctrl_BackPath_near);
drv_ctrl_BackPath_far := POU_interlock.out_ctrl_1;

// NETWORK 26
//   KM13: Module_1 : | AT %IX5.1
//   var_KL13: KM13; электродвигатель тросового толкателя обгонного пути
//   var_KL14: KM13; электродвигатель тросового толкателя обгонного пути (реверс)
_w3 := drv_ctrl_BackPath_far AND NOT lim_BackPath_far AND KM13;
var_KL13 := _w3;
var_KL14 R= _w3;

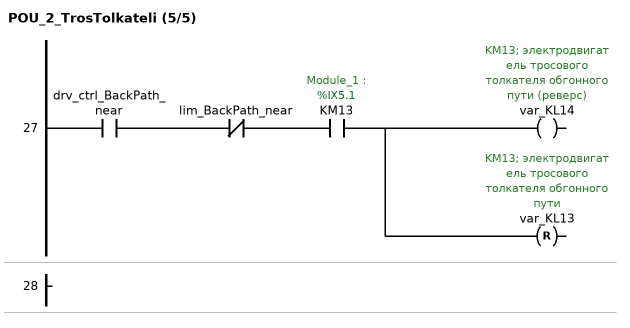
// NETWORK 27
//   KM13: Module_1 : | AT %IX5.1
//   var_KL14: KM13; электродвигатель тросового толкателя обгонного пути (реверс)
//   var_KL13: KM13; электродвигатель тросового толкателя обгонного пути
_w4 := drv_ctrl_BackPath_near AND NOT lim_BackPath_near AND KM13;
var_KL14 := _w4;
var_KL13 R= _w4;

// NETWORK 28

END_PROGRAM

// MyController/Application/POU_interlock_double
PROGRAM POU_interlock_double
VAR_INPUT
	in_post_ctrl_1: BOOL;
	in_post_ctrl_2: BOOL;
	in_prog_ctrl_1: BOOL;
	in_prog_ctrl_2: BOOL;
END_VAR

VAR
	out_post_ctrl_2: BOOL;
	out_post_ctrl_1: BOOL;
	out_prog_ctrl_1: BOOL;
	out_prog_ctrl_2: BOOL;
END_VAR
VAR_OUTPUT
	out_sum_ctrl_1: BOOL;
	out_sum_ctrl_2: BOOL;
END_VAR

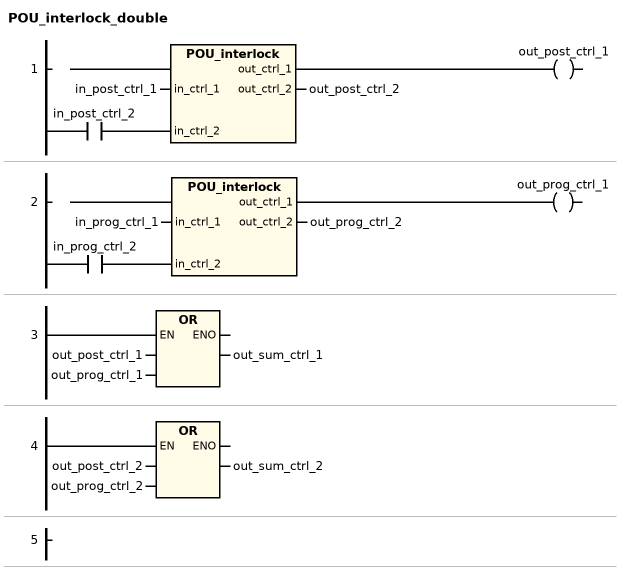
// NETWORK 1
POU_interlock(in_ctrl_1 := in_post_ctrl_1, in_ctrl_2 := in_post_ctrl_2, out_ctrl_2 => out_post_ctrl_2);
out_post_ctrl_1 := POU_interlock.out_ctrl_1;

// NETWORK 2
POU_interlock(in_ctrl_1 := in_prog_ctrl_1, in_ctrl_2 := in_prog_ctrl_2, out_ctrl_2 => out_prog_ctrl_2);
out_prog_ctrl_1 := POU_interlock.out_ctrl_1;

// NETWORK 3
out_sum_ctrl_1 := out_post_ctrl_1 OR out_prog_ctrl_1;

// NETWORK 4
out_sum_ctrl_2 := out_post_ctrl_2 OR out_prog_ctrl_2;

// NETWORK 5

END_PROGRAM

// MyController/Application/POU_interlock
PROGRAM POU_interlock
VAR
	err_ctrl: BOOL;
END_VAR
VAR_INPUT
	in_ctrl_1: BOOL;
END_VAR
VAR_OUTPUT
	out_ctrl_1: BOOL;
END_VAR
VAR_INPUT
	in_ctrl_2: BOOL;
END_VAR
VAR_OUTPUT
	out_ctrl_2: BOOL;
END_VAR

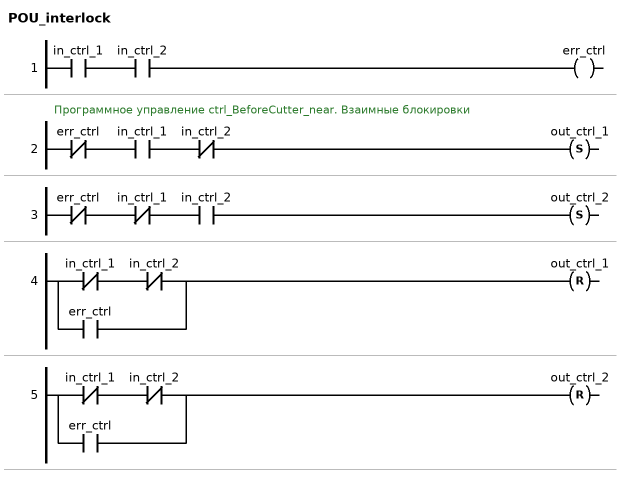
// NETWORK 1
err_ctrl := in_ctrl_1 AND in_ctrl_2;

// NETWORK 2
// Программное управление ctrl_BeforeCutter_near. Взаимные блокировки
out_ctrl_1 S= NOT err_ctrl AND in_ctrl_1 AND NOT in_ctrl_2;

// NETWORK 3
out_ctrl_2 S= NOT err_ctrl AND NOT in_ctrl_1 AND in_ctrl_2;

// NETWORK 4
out_ctrl_1 R= NOT in_ctrl_1 AND NOT in_ctrl_2 OR err_ctrl;

// NETWORK 5
out_ctrl_2 R= NOT in_ctrl_1 AND NOT in_ctrl_2 OR err_ctrl;

END_PROGRAM

// MyController/Application/POU_9_altivars
PROGRAM POU_9_altivars
VAR
	altivar_0: Altivar71_Control;
END_VAR
VAR_INPUT
	var_Altivar_0_en: BOOL;
	var_Altivar_0_freq: INT;
	var_Altivar_0_fwd: BOOL;
	var_Altivar_0_rev: BOOL;
END_VAR
VAR
	altivar_1: Altivar71_Control;
END_VAR
VAR_INPUT
	var_Altivar_1_en: BOOL;
	var_Altivar_1_freq: INT;
	var_Altivar_1_fwd: BOOL;
	var_Altivar_1_rev: BOOL;
END_VAR
VAR
	altivar_2: Altivar71_Control;
END_VAR
VAR_INPUT
	var_Altivar_2_en: BOOL;
	var_Altivar_2_freq: INT;
	var_Altivar_2_fwd: BOOL;
	var_Altivar_2_rev: BOOL;
END_VAR

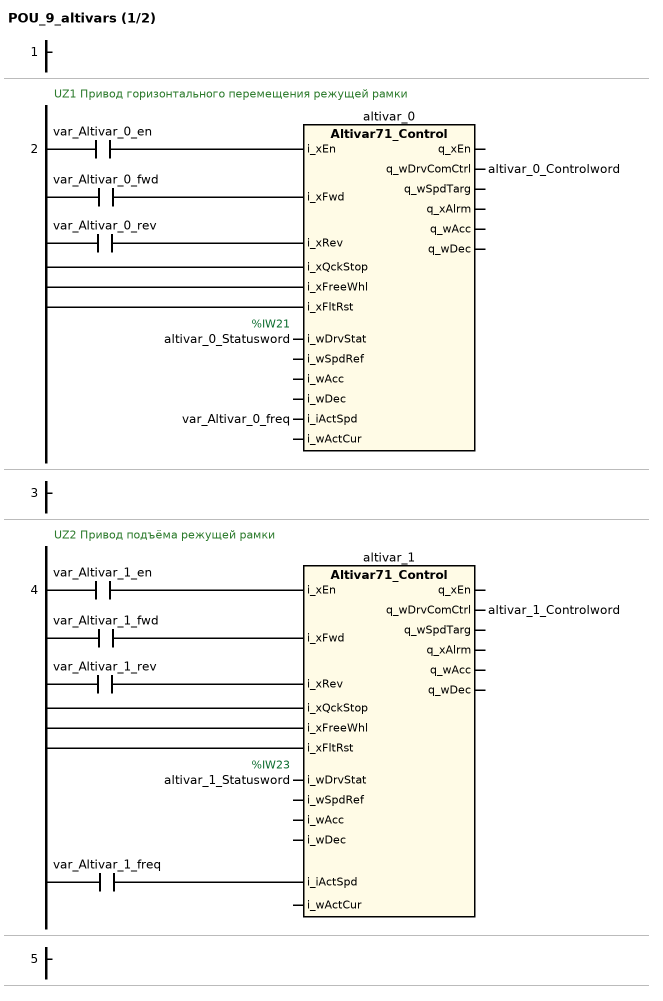
// NETWORK 1

// NETWORK 2
// UZ1 Привод горизонтального перемещения режущей рамки
//   altivar_0_Statusword: Altivar_71_0 : | AT %IW21
//   altivar_0_Controlword: Altivar_71_0 : | AT %QW18
altivar_0(
    i_xEn := var_Altivar_0_en,
    i_xFwd := var_Altivar_0_fwd,
    i_xRev := var_Altivar_0_rev,
    i_xQckStop := TRUE,
    i_xFreeWhl := TRUE,
    i_xFltRst := TRUE,
    i_wDrvStat := altivar_0_Statusword,
    i_iActSpd := var_Altivar_0_freq,
    q_wDrvComCtrl => altivar_0_Controlword); // Altivar71_Control

// NETWORK 3

// NETWORK 4
// UZ2 Привод подъёма режущей рамки
//   altivar_1_Statusword: Altivar_71_1 : | AT %IW23
//   altivar_1_Controlword: Altivar_71_1 : | AT %QW22
altivar_1(
    i_xEn := var_Altivar_1_en,
    i_xFwd := var_Altivar_1_fwd,
    i_xRev := var_Altivar_1_rev,
    i_xQckStop := TRUE,
    i_xFreeWhl := TRUE,
    i_xFltRst := TRUE,
    i_wDrvStat := altivar_1_Statusword,
    i_iActSpd := var_Altivar_1_freq,
    q_wDrvComCtrl => altivar_1_Controlword); // Altivar71_Control

// NETWORK 5

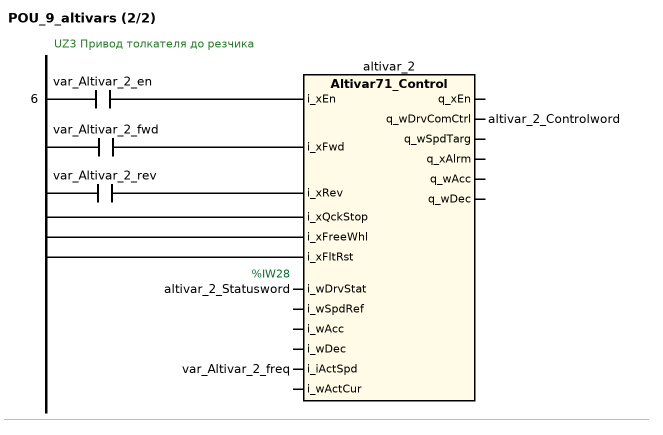
// NETWORK 6
// UZ3 Привод толкателя до резчика
//   altivar_2_Statusword: Altivar_71_2 : | AT %IW28
//   altivar_2_Controlword: Altivar_71_2 : | AT %QW24
altivar_2(
    i_xEn := var_Altivar_2_en,
    i_xFwd := var_Altivar_2_fwd,
    i_xRev := var_Altivar_2_rev,
    i_xQckStop := TRUE,
    i_xFreeWhl := TRUE,
    i_xFltRst := TRUE,
    i_wDrvStat := altivar_2_Statusword,
    i_iActSpd := var_Altivar_2_freq,
    q_wDrvComCtrl => altivar_2_Controlword); // Altivar71_Control

END_PROGRAM

// MyController/Application/POU_3_PodvodTelezhki
PROGRAM POU_3_PodvodTelezhki
VAR
	sens_Troll_is: BOOL := FALSE;
	step_CentrTroll_INIT: BOOL := TRUE;
	ctrl_CentrTroll_in: BOOL;
	sens_CentrTroll_in: BOOL;
	step_CentrTroll_in_EXEC: BOOL;
	step_CentrTroll_in_OVER: BOOL;
	step_CentrTroll_in_ERR: BOOL;
	timer_CentrTroll_in: TIME;
	ctrl_CentrTroll_out: BOOL;
	sens_CentrTroll_out: BOOL;
	step_CentrTroll_out_EXEC: BOOL;
	step_CentrTroll_out_OVER: BOOL;
	step_CentrTroll_out_ERR: BOOL;
END_VAR

VAR
	timer_CentrTroll_out: TIME;
END_VAR

